LIN {X 0,Y 309.454,Z 977.493,A -85,B 0,C 180,E1 27160.011,E2 27160.011} C_VEL
LIN {X 0,Y 310.124,Z 964.953,A -85,B 0,C 180,E1 27165.897,E2 27165.897} C_VEL
LIN {X 0,Y 310.342,Z 957.233,A -85,B 0,C 180,E1 27171.598,E2 27171.598} C_VEL
LIN {X 0,Y 311.292,Z 953.109,A -85,B 0,C 180,E1 27177.214,E2 27177.214} C_VEL
LIN {X 0,Y 311.401,Z 954.291,A -85,B 0,C 180,E1 27181.386,E2 27181.386} C_VEL
LIN {X 0,Y 311.732,Z 959.799,A -85,B 0,C 180,E1 27186.955,E2 27186.955} C_VEL
LIN {X 0,Y 312.391,Z 969.833,A -85,B 0,C 180,E1 27192.716,E2 27192.716} C_VEL
LIN {X 0,Y 312.414,Z 984.77,A -85,B 0,C 180,E1 27198.53,E2 27198.53} C_VEL
LIN {X 0,Y 312.191,Z 989.255,A -85,B 0,C 180,E1 27199.981,E2 27199.981} C_VEL
LIN {X 0,Y 287.34,Z 1027.158,A -85,B 0,C 180,E1 27203.968,E2 27203.968} C_VEL
LIN {X 0,Y 260.3,Z 1061.028,A -85,B 0,C 180,E1 27209.446,E2 27209.446} C_VEL
LIN {X 0,Y 233.843,Z 1089.665,A -85,B 0,C 180,E1 27216.897,E2 27216.897} C_VEL
LIN {X 0,Y 212.045,Z 1111.278,A -85,B 0,C 180,E1 27225.984,E2 27225.984} C_VEL
LIN {X 0,Y 195.512,Z 1127.849,A -85,B 0,C 180,E1 27237.243,E2 27237.243} C_VEL
LIN {X 0,Y 185.737,Z 1139.665,A -85,B 0,C 180,E1 27251.006,E2 27251.006} C_VEL
LIN {X 0,Y 183.31,Z 1144.428,A -85,B 0,C 180,E1 27261.462,E2 27261.462} C_VEL
LIN {X 0,Y 183.515,Z 1145.902,A -85,B 0,C 180,E1 27269.997,E2 27269.997} C_VEL
LIN {X 0,Y 183.436,Z 1145.117,A -85,B 0,C 180,E1 27279.48,E2 27279.48} C_VEL
LIN {X 0,Y 186.512,Z 1140.958,A -85,B 0,C 180,E1 27290.599,E2 27290.599} C_VEL
LIN {X 0,Y 197.046,Z 1130.929,A -85,B 0,C 180,E1 27303.776,E2 27303.776} C_VEL
LIN {X 0,Y 217.166,Z 1113.725,A -85,B 0,C 180,E1 27316.111,E2 27316.111} C_VEL
LIN {X 0,Y 243.736,Z 1090.221,A -85,B 0,C 180,E1 27325.671,E2 27325.671} C_VEL
LIN {X 0,Y 272.358,Z 1061.63,A -85,B 0,C 180,E1 27332.584,E2 27332.584} C_VEL
LIN {X 0,Y 300.342,Z 1028.677,A -85,B 0,C 180,E1 27337.531,E2 27337.531} C_VEL
LIN {X 0,Y 320.87,Z 1000.29,A -85,B 0,C 180,E1 27340.365,E2 27340.365} C_VEL
LIN {X 0,Y 321.893,Z 993.539,A -85,B 0,C 180,E1 27342.656,E2 27342.656} C_VEL
LIN {X 0,Y 322.199,Z 981.849,A -85,B 0,C 180,E1 27348.504,E2 27348.504} C_VEL
LIN {X 0,Y 322.094,Z 974.677,A -85,B 0,C 180,E1 27354.621,E2 27354.621} C_VEL
LIN {X 0,Y 322.235,Z 972.945,A -85,B 0,C 180,E1 27357.317,E2 27357.317} C_VEL
LIN {X 0,Y 322.11,Z 972.654,A -85,B 0,C 180,E1 27360.004,E2 27360.004} C_VEL
LIN {X 0,Y 320.931,Z 976.591,A -85,B 0,C 180,E1 27365.407,E2 27365.407} C_VEL
LIN {X 0,Y 319.909,Z 984.239,A -85,B 0,C 180,E1 27370.893,E2 27370.893} C_VEL
LIN {X 0,Y 318.076,Z 996.337,A -85,B 0,C 180,E1 27376.563,E2 27376.563} C_VEL
LIN {X 0,Y 317.265,Z 1000.211,A -85,B 0,C 180,E1 27378.034,E2 27378.034} C_VEL
LIN {X 0,Y 295.491,Z 1029.491,A -85,B 0,C 180,E1 27381.587,E2 27381.587} C_VEL
LIN {X 0,Y 267.613,Z 1060.339,A -85,B 0,C 180,E1 27386.963,E2 27386.963} C_VEL
LIN {X 0,Y 241.205,Z 1085.273,A -85,B 0,C 180,E1 27393.896,E2 27393.896} C_VEL
LIN {X 0,Y 219.023,Z 1103.942,A -85,B 0,C 180,E1 27402.129,E2 27402.129} C_VEL
LIN {X 0,Y 199.19,Z 1119.649,A -85,B 0,C 180,E1 27413.993,E2 27413.993} C_VEL
LIN {X 0,Y 196.821,Z 1121.44,A -85,B 0,C 180,E1 27415.996,E2 27415.996} C_VEL
LIN {X 0,Y 188.409,Z 1125.457,A -85,B 0,C 180,E1 27420.414,E2 27420.414} C_VEL
LIN {X 0,Y 180.821,Z 1128.688,A -85,B 0,C 180,E1 27425.237,E2 27425.237} C_VEL
LIN {X 0,Y 176.46,Z 1132.191,A -85,B 0,C 180,E1 27435.117,E2 27435.117} C_VEL
LIN {X 0,Y 175.258,Z 1133.272,A -85,B 0,C 180,E1 27445.057,E2 27445.057} C_VEL
LIN {X 0,Y 176.038,Z 1131.933,A -85,B 0,C 180,E1 27454.927,E2 27454.927} C_VEL
LIN {X 0,Y 179.788,Z 1126.98,A -85,B 0,C 180,E1 27467.111,E2 27467.111} C_VEL
LIN {X 0,Y 191.399,Z 1115.835,A -85,B 0,C 180,E1 27480.879,E2 27480.879} C_VEL
LIN {X 0,Y 209.17,Z 1100.079,A -85,B 0,C 180,E1 27491.935,E2 27491.935} C_VEL
LIN {X 0,Y 231.682,Z 1079.475,A -85,B 0,C 180,E1 27500.765,E2 27500.765} C_VEL
LIN {X 0,Y 258.39,Z 1052.11,A -85,B 0,C 180,E1 27507.992,E2 27507.992} C_VEL
LIN {X 0,Y 285.416,Z 1019.388,A -85,B 0,C 180,E1 27513.41,E2 27513.41} C_VEL
LIN {X 0,Y 302.07,Z 995.756,A -85,B 0,C 180,E1 27516.102,E2 27516.102} C_VEL
LIN {X 0,Y 304.033,Z 986.317,A -85,B 0,C 180,E1 27519.215,E2 27519.215} C_VEL
LIN {X 0,Y 305.429,Z 973.42,A -85,B 0,C 180,E1 27524.943,E2 27524.943} C_VEL
LIN {X 0,Y 306.041,Z 964.764,A -85,B 0,C 180,E1 27530.947,E2 27530.947} C_VEL
LIN {X 0,Y 307.174,Z 959.952,A -85,B 0,C 180,E1 27537.176,E2 27537.176} C_VEL
LIN {X 0,Y 307.282,Z 961.092,A -85,B 0,C 180,E1 27541.404,E2 27541.404} C_VEL
LIN {X 0,Y 307.545,Z 967.728,A -85,B 0,C 180,E1 27547.76,E2 27547.76} C_VEL
LIN {X 0,Y 307.681,Z 978.547,A -85,B 0,C 180,E1 27553.56,E2 27553.56} C_VEL
LIN {X 0,Y 307.106,Z 992.03,A -85,B 0,C 180,E1 27558.702,E2 27558.702} C_VEL
LIN {X 0,Y 305.015,Z 996.226,A -85,B 0,C 180,E1 27559.302,E2 27559.302} C_VEL
LIN {X 0,Y 282.523,Z 1028.725,A -85,B 0,C 180,E1 27562.74,E2 27562.74} C_VEL
LIN {X 0,Y 256.385,Z 1060.564,A -85,B 0,C 180,E1 27567.857,E2 27567.857} C_VEL
LIN {X 0,Y 228.987,Z 1089.241,A -85,B 0,C 180,E1 27575.247,E2 27575.247} C_VEL
LIN {X 0,Y 206.22,Z 1110.893,A -85,B 0,C 180,E1 27584.399,E2 27584.399} C_VEL
LIN {X 0,Y 188.676,Z 1127.497,A -85,B 0,C 180,E1 27595.897,E2 27595.897} C_VEL
LIN {X 0,Y 178.135,Z 1139.34,A -85,B 0,C 180,E1 27610.162,E2 27610.162} C_VEL
LIN {X 0,Y 175.558,Z 1143.769,A -85,B 0,C 180,E1 27620.084,E2 27620.084} C_VEL
LIN {X 0,Y 175.605,Z 1145.616,A -85,B 0,C 180,E1 27629.997,E2 27629.997} C_VEL
LIN {X 0,Y 175.561,Z 1144.846,A -85,B 0,C 180,E1 27639.91,E2 27639.91} C_VEL
LIN {X 0,Y 179.205,Z 1140.454,A -85,B 0,C 180,E1 27651.988,E2 27651.988} C_VEL
LIN {X 0,Y 190.306,Z 1130.7,A -85,B 0,C 180,E1 27665.144,E2 27665.144} C_VEL
LIN {X 0,Y 210.651,Z 1114.288,A -85,B 0,C 180,E1 27677.288,E2 27677.288} C_VEL
LIN {X 0,Y 237.393,Z 1091.652,A -85,B 0,C 180,E1 27686.769,E2 27686.769} C_VEL
LIN {X 0,Y 265.849,Z 1064.402,A -85,B 0,C 180,E1 27693.552,E2 27693.552} C_VEL
LIN {X 0,Y 292.81,Z 1034.247,A -85,B 0,C 180,E1 27698.264,E2 27698.264} C_VEL
LIN {X 0,Y 316.359,Z 1002.822,A -85,B 0,C 180,E1 27701.561,E2 27701.561} C_VEL
LIN {X 0,Y 317.281,Z 991.089,A -85,B 0,C 180,E1 27706.932,E2 27706.932} C_VEL
LIN {X 0,Y 317.494,Z 984.09,A -85,B 0,C 180,E1 27711.797,E2 27711.797} C_VEL
LIN {X 0,Y 317.754,Z 979.539,A -85,B 0,C 180,E1 27717.279,E2 27717.279} C_VEL
LIN {X 0,Y 317.364,Z 979.71,A -85,B 0,C 180,E1 27720.922,E2 27720.922} C_VEL
LIN {X 0,Y 315.966,Z 984.954,A -85,B 0,C 180,E1 27727.008,E2 27727.008} C_VEL
LIN {X 0,Y 314.446,Z 993.783,A -85,B 0,C 180,E1 27732.491,E2 27732.491} C_VEL
LIN {X 0,Y 312.348,Z 1003.618,A -85,B 0,C 180,E1 27736.876,E2 27736.876} C_VEL
LIN {X 0,Y 310.356,Z 1006.988,A -85,B 0,C 180,E1 27737.456,E2 27737.456} C_VEL
LIN {X 0,Y 281.848,Z 1041.952,A -85,B 0,C 180,E1 27741.953,E2 27741.953} C_VEL
LIN {X 0,Y 251.952,Z 1072.057,A -85,B 0,C 180,E1 27748.147,E2 27748.147} C_VEL
LIN {X 0,Y 224.69,Z 1095.458,A -85,B 0,C 180,E1 27756.196,E2 27756.196} C_VEL
LIN {X 0,Y 201.8,Z 1112.987,A -85,B 0,C 180,E1 27766.417,E2 27766.417} C_VEL
LIN {X 0,Y 186.729,Z 1124.294,A -85,B 0,C 180,E1 27777.828,E2 27777.828} C_VEL
LIN {X 0,Y 180.821,Z 1128.688,A -85,B 0,C 180,E1 27785.237,E2 27785.237} C_VEL
LIN {X 0,Y 176.154,Z 1130.599,A -85,B 0,C 180,E1 27789.115,E2 27789.115} C_VEL
LIN {X 0,Y 168.559,Z 1132.598,A -85,B 0,C 180,E1 27795.169,E2 27795.169} C_VEL
LIN {X 0,Y 168.269,Z 1132.704,A -85,B 0,C 180,E1 27795.909,E2 27795.909} C_VEL
LIN {X 0,Y 167.345,Z 1133.56,A -85,B 0,C 180,E1 27804.822,E2 27804.822} C_VEL
LIN {X 0,Y 168.161,Z 1132.229,A -85,B 0,C 180,E1 27815.159,E2 27815.159} C_VEL
LIN {X 0,Y 172.214,Z 1127.308,A -85,B 0,C 180,E1 27827.888,E2 27827.888} C_VEL
LIN {X 0,Y 184.575,Z 1116.187,A -85,B 0,C 180,E1 27842.154,E2 27842.154} C_VEL
LIN {X 0,Y 203.287,Z 1100.465,A -85,B 0,C 180,E1 27853.443,E2 27853.443} C_VEL
LIN {X 0,Y 226.708,Z 1079.898,A -85,B 0,C 180,E1 27862.331,E2 27862.331} C_VEL
LIN {X 0,Y 253.939,Z 1052.898,A -85,B 0,C 180,E1 27869.445,E2 27869.445} C_VEL
LIN {X 0,Y 281.772,Z 1020.113,A -85,B 0,C 180,E1 27874.823,E2 27874.823} C_VEL
LIN {X 0,Y 297.696,Z 997.877,A -85,B 0,C 180,E1 27877.424,E2 27877.424} C_VEL
LIN {X 0,Y 300.165,Z 983.944,A -85,B 0,C 180,E1 27883.045,E2 27883.045} C_VEL
LIN {X 0,Y 301.3,Z 974.505,A -85,B 0,C 180,E1 27888.425,E2 27888.425} C_VEL
LIN {X 0,Y 302.298,Z 968.507,A -85,B 0,C 180,E1 27894.259,E2 27894.259} C_VEL
LIN {X 0,Y 302.991,Z 966.741,A -85,B 0,C 180,E1 27897.137,E2 27897.137} C_VEL
LIN {X 0,Y 303.1,Z 967.874,A -85,B 0,C 180,E1 27901.424,E2 27901.424} C_VEL
LIN {X 0,Y 303.108,Z 974.62,A -85,B 0,C 180,E1 27907.874,E2 27907.874} C_VEL
LIN {X 0,Y 302.846,Z 985.681,A -85,B 0,C 180,E1 27913.703,E2 27913.703} C_VEL
LIN {X 0,Y 301.796,Z 996.683,A -85,B 0,C 180,E1 27917.943,E2 27917.943} C_VEL
LIN {X 0,Y 277.843,Z 1030.29,A -85,B 0,C 180,E1 27921.47,E2 27921.47} C_VEL
LIN {X 0,Y 250.98,Z 1061.929,A -85,B 0,C 180,E1 27926.585,E2 27926.585} C_VEL
LIN {X 0,Y 223.105,Z 1090.047,A -85,B 0,C 180,E1 27933.928,E2 27933.928} C_VEL
LIN {X 0,Y 197.761,Z 1113.049,A -85,B 0,C 180,E1 27944.125,E2 27944.125} C_VEL
LIN {X 0,Y 179.941,Z 1129.015,A -85,B 0,C 180,E1 27956.302,E2 27956.302} C_VEL
LIN {X 0,Y 170.58,Z 1139.013,A -85,B 0,C 180,E1 27969.244,E2 27969.244} C_VEL
LIN {X 0,Y 167.367,Z 1144.369,A -85,B 0,C 180,E1 27983.143,E2 27983.143} C_VEL
LIN {X 0,Y 167.695,Z 1145.33,A -85,B 0,C 180,E1 27989.997,E2 27989.997} C_VEL
LIN {X 0,Y 167.704,Z 1144.576,A -85,B 0,C 180,E1 28000.379,E2 28000.379} C_VEL
LIN {X 0,Y 173.437,Z 1138.737,A -85,B 0,C 180,E1 28015.823,E2 28015.823} C_VEL
LIN {X 0,Y 188.304,Z 1126.942,A -85,B 0,C 180,E1 28029.936,E2 28029.936} C_VEL
LIN {X 0,Y 209.62,Z 1110.564,A -85,B 0,C 180,E1 28040.796,E2 28040.796} C_VEL
LIN {X 0,Y 236.369,Z 1088.569,A -85,B 0,C 180,E1 28049.353,E2 28049.353} C_VEL
LIN {X 0,Y 266.452,Z 1060.199,A -85,B 0,C 180,E1 28055.909,E2 28055.909} C_VEL
LIN {X 0,Y 296.399,Z 1026.341,A -85,B 0,C 180,E1 28060.667,E2 28060.667} C_VEL
LIN {X 0,Y 311.26,Z 1006.345,A -85,B 0,C 180,E1 28062.709,E2 28062.709} C_VEL
LIN {X 0,Y 312.419,Z 995.821,A -85,B 0,C 180,E1 28067.932,E2 28067.932} C_VEL
LIN {X 0,Y 312.75,Z 989.184,A -85,B 0,C 180,E1 28073.068,E2 28073.068} C_VEL
LIN {X 0,Y 313.176,Z 986.028,A -85,B 0,C 180,E1 28077.239,E2 28077.239} C_VEL
LIN {X 0,Y 313.053,Z 985.699,A -85,B 0,C 180,E1 28080.004,E2 28080.004} C_VEL
LIN {X 0,Y 311.462,Z 989.786,A -85,B 0,C 180,E1 28085.572,E2 28085.572} C_VEL
LIN {X 0,Y 309.922,Z 996.772,A -85,B 0,C 180,E1 28090.639,E2 28090.639} C_VEL
LIN {X 0,Y 307.308,Z 1007.696,A -85,B 0,C 180,E1 28095.956,E2 28095.956} C_VEL
LIN {X 0,Y 279.608,Z 1041.247,A -85,B 0,C 180,E1 28100.273,E2 28100.273} C_VEL
LIN {X 0,Y 249.573,Z 1070.924,A -85,B 0,C 180,E1 28106.175,E2 28106.175} C_VEL
LIN {X 0,Y 221.618,Z 1094.277,A -85,B 0,C 180,E1 28113.878,E2 28113.878} C_VEL
LIN {X 0,Y 199.18,Z 1110.983,A -85,B 0,C 180,E1 28123.062,E2 28123.062} C_VEL
LIN {X 0,Y 179.996,Z 1124.437,A -85,B 0,C 180,E1 28136.312,E2 28136.312} C_VEL
LIN {X 0,Y 170.661,Z 1131.02,A -85,B 0,C 180,E1 28149.26,E2 28149.26} C_VEL
LIN {X 0,Y 168.269,Z 1132.704,A -85,B 0,C 180,E1 28155.909,E2 28155.909} C_VEL
LIN {X 0,Y 164.949,Z 1133.468,A -85,B 0,C 180,E1 28160.259,E2 28160.259} C_VEL
LIN {X 0,Y 159.505,Z 1133.688,A -85,B 0,C 180,E1 28167.01,E2 28167.01} C_VEL
LIN {X 0,Y 159.476,Z 1133.631,A -85,B 0,C 180,E1 28167.801,E2 28167.801} C_VEL
LIN {X 0,Y 160.307,Z 1132.525,A -85,B 0,C 180,E1 28175.412,E2 28175.412} C_VEL
LIN {X 0,Y 164.681,Z 1127.635,A -85,B 0,C 180,E1 28188.736,E2 28188.736} C_VEL
LIN {X 0,Y 177.847,Z 1116.538,A -85,B 0,C 180,E1 28203.527,E2 28203.527} C_VEL
LIN {X 0,Y 197.547,Z 1100.85,A -85,B 0,C 180,E1 28215.041,E2 28215.041} C_VEL
LIN {X 0,Y 223.181,Z 1079.148,A -85,B 0,C 180,E1 28224.344,E2 28224.344} C_VEL
LIN {X 0,Y 251.638,Z 1051.584,A -85,B 0,C 180,E1 28231.376,E2 28231.376} C_VEL
LIN {X 0,Y 280.049,Z 1018.714,A -85,B 0,C 180,E1 28236.538,E2 28236.538} C_VEL
LIN {X 0,Y 292.521,Z 1001.831,A -85,B 0,C 180,E1 28238.415,E2 28238.415} C_VEL
LIN {X 0,Y 295.236,Z 989.526,A -85,B 0,C 180,E1 28243.545,E2 28243.545} C_VEL
LIN {X 0,Y 296.655,Z 981.453,A -85,B 0,C 180,E1 28248.241,E2 28248.241} C_VEL
LIN {X 0,Y 297.788,Z 975.178,A -85,B 0,C 180,E1 28254.172,E2 28254.172} C_VEL
LIN {X 0,Y 298.613,Z 973.397,A -85,B 0,C 180,E1 28257.095,E2 28257.095} C_VEL
LIN {X 0,Y 298.705,Z 974.518,A -85,B 0,C 180,E1 28261.445,E2 28261.445} C_VEL
LIN {X 0,Y 298.49,Z 981.466,A -85,B 0,C 180,E1 28267.997,E2 28267.997} C_VEL
LIN {X 0,Y 297.701,Z 992.509,A -85,B 0,C 180,E1 28273.806,E2 28273.806} C_VEL
LIN {X 0,Y 296.878,Z 999.978,A -85,B 0,C 180,E1 28276.765,E2 28276.765} C_VEL
LIN {X 0,Y 268.977,Z 1037.272,A -85,B 0,C 180,E1 28280.878,E2 28280.878} C_VEL
LIN {X 0,Y 240.531,Z 1068.562,A -85,B 0,C 180,E1 28286.402,E2 28286.402} C_VEL
LIN {X 0,Y 214.164,Z 1093.626,A -85,B 0,C 180,E1 28293.59,E2 28293.59} C_VEL
LIN {X 0,Y 190.431,Z 1114.141,A -85,B 0,C 180,E1 28303.245,E2 28303.245} C_VEL
LIN {X 0,Y 171.503,Z 1130.225,A -85,B 0,C 180,E1 28316.419,E2 28316.419} C_VEL
LIN {X 0,Y 161.893,Z 1139.987,A -85,B 0,C 180,E1 28330.929,E2 28330.929} C_VEL
LIN {X 0,Y 159.495,Z 1144.421,A -85,B 0,C 180,E1 28344.56,E2 28344.56} C_VEL
LIN {X 0,Y 159.797,Z 1145.045,A -85,B 0,C 180,E1 28349.997,E2 28349.997} C_VEL
LIN {X 0,Y 159.842,Z 1144.304,A -85,B 0,C 180,E1 28360.896,E2 28360.896} C_VEL
LIN {X 0,Y 166.167,Z 1138.49,A -85,B 0,C 180,E1 28377.042,E2 28377.042} C_VEL
LIN {X 0,Y 183.695,Z 1125.645,A -85,B 0,C 180,E1 28392.573,E2 28392.573} C_VEL
LIN {X 0,Y 209.582,Z 1106.659,A -85,B 0,C 180,E1 28404.386,E2 28404.386} C_VEL
LIN {X 0,Y 239.72,Z 1082.029,A -85,B 0,C 180,E1 28412.847,E2 28412.847} C_VEL
LIN {X 0,Y 269.467,Z 1053.611,A -85,B 0,C 180,E1 28418.583,E2 28418.583} C_VEL
LIN {X 0,Y 296.724,Z 1022.644,A -85,B 0,C 180,E1 28422.514,E2 28422.514} C_VEL
LIN {X 0,Y 306.171,Z 1010.273,A -85,B 0,C 180,E1 28423.751,E2 28423.751} C_VEL
LIN {X 0,Y 307.598,Z 1000.079,A -85,B 0,C 180,E1 28429.262,E2 28429.262} C_VEL
LIN {X 0,Y 308.074,Z 994.353,A -85,B 0,C 180,E1 28434.376,E2 28434.376} C_VEL
LIN {X 0,Y 308.402,Z 992.413,A -85,B 0,C 180,E1 28437.196,E2 28437.196} C_VEL
LIN {X 0,Y 308.295,Z 992.056,A -85,B 0,C 180,E1 28440.004,E2 28440.004} C_VEL
LIN {X 0,Y 306.568,Z 996.274,A -85,B 0,C 180,E1 28445.661,E2 28445.661} C_VEL
LIN {X 0,Y 304.544,Z 1003.435,A -85,B 0,C 180,E1 28450.829,E2 28450.829} C_VEL
LIN {X 0,Y 302.291,Z 1011.366,A -85,B 0,C 180,E1 28454.846,E2 28454.846} C_VEL
LIN {X 0,Y 275.542,Z 1042.801,A -85,B 0,C 180,E1 28458.919,E2 28458.919} C_VEL
LIN {X 0,Y 244.948,Z 1072.087,A -85,B 0,C 180,E1 28464.72,E2 28464.72} C_VEL
LIN {X 0,Y 215.386,Z 1095.811,A -85,B 0,C 180,E1 28472.663,E2 28472.663} C_VEL
LIN {X 0,Y 191.129,Z 1112.845,A -85,B 0,C 180,E1 28482.57,E2 28482.57} C_VEL
LIN {X 0,Y 171.669,Z 1125.654,A -85,B 0,C 180,E1 28496.367,E2 28496.367} C_VEL
LIN {X 0,Y 163.133,Z 1131.282,A -85,B 0,C 180,E1 28508.256,E2 28508.256} C_VEL
LIN {X 0,Y 159.816,Z 1133.583,A -85,B 0,C 180,E1 28519.103,E2 28519.103} C_VEL
LIN {X 0,Y 159.476,Z 1133.631,A -85,B 0,C 180,E1 28527.801,E2 28527.801} C_VEL
LIN {X 0,Y 157.366,Z 1133.201,A -85,B 0,C 180,E1 28532.48,E2 28532.48} C_VEL
LIN {X 0,Y 153.389,Z 1131.539,A -85,B 0,C 180,E1 28540.523,E2 28540.523} C_VEL
LIN {X 0,Y 160.85,Z 1124.949,A -85,B 0,C 180,E1 28555.012,E2 28555.012} C_VEL
LIN {X 0,Y 179.309,Z 1110.927,A -85,B 0,C 180,E1 28570.312,E2 28570.312} C_VEL
LIN {X 0,Y 204.992,Z 1091.025,A -85,B 0,C 180,E1 28581.773,E2 28581.773} C_VEL
LIN {X 0,Y 233.615,Z 1066.025,A -85,B 0,C 180,E1 28589.903,E2 28589.903} C_VEL
LIN {X 0,Y 261.479,Z 1037.424,A -85,B 0,C 180,E1 28595.538,E2 28595.538} C_VEL
LIN {X 0,Y 287.755,Z 1004.894,A -85,B 0,C 180,E1 28599.73,E2 28599.73} C_VEL
LIN {X 0,Y 290.688,Z 993.375,A -85,B 0,C 180,E1 28604.933,E2 28604.933} C_VEL
LIN {X 0,Y 292.054,Z 986.379,A -85,B 0,C 180,E1 28609.452,E2 28609.452} C_VEL
LIN {X 0,Y 293.263,Z 981.857,A -85,B 0,C 180,E1 28614.081,E2 28614.081} C_VEL
LIN {X 0,Y 294.123,Z 979.999,A -85,B 0,C 180,E1 28617.051,E2 28617.051} C_VEL
LIN {X 0,Y 294.203,Z 981.13,A -85,B 0,C 180,E1 28621.467,E2 28621.467} C_VEL
LIN {X 0,Y 293.788,Z 987.176,A -85,B 0,C 180,E1 28627.382,E2 28627.382} C_VEL
LIN {X 0,Y 292.679,Z 997.658,A -85,B 0,C 180,E1 28633.146,E2 28633.146} C_VEL
LIN {X 0,Y 291.155,Z 1004.413,A -85,B 0,C 180,E1 28635.725,E2 28635.725} C_VEL
LIN {X 0,Y 264.513,Z 1038.724,A -85,B 0,C 180,E1 28639.505,E2 28639.505} C_VEL
LIN {X 0,Y 234.012,Z 1071.132,A -85,B 0,C 180,E1 28645.301,E2 28645.301} C_VEL
LIN {X 0,Y 204.459,Z 1097.801,A -85,B 0,C 180,E1 28653.445,E2 28653.445} C_VEL
LIN {X 0,Y 179.421,Z 1118.05,A -85,B 0,C 180,E1 28664.281,E2 28664.281} C_VEL
LIN {X 0,Y 163.219,Z 1131.213,A -85,B 0,C 180,E1 28676.403,E2 28676.403} C_VEL
LIN {X 0,Y 153.311,Z 1140.929,A -85,B 0,C 180,E1 28692.797,E2 28692.797} C_VEL
LIN {X 0,Y 151.573,Z 1144.313,A -85,B 0,C 180,E1 28705.293,E2 28705.293} C_VEL
LIN {X 0,Y 151.885,Z 1144.758,A -85,B 0,C 180,E1 28709.997,E2 28709.997} C_VEL
LIN {X 0,Y 151.992,Z 1144.033,A -85,B 0,C 180,E1 28721.466,E2 28721.466} C_VEL
LIN {X 0,Y 158.972,Z 1138.242,A -85,B 0,C 180,E1 28738.374,E2 28738.374} C_VEL
LIN {X 0,Y 177.932,Z 1125.291,A -85,B 0,C 180,E1 28754.474,E2 28754.474} C_VEL
LIN {X 0,Y 204.928,Z 1106.462,A -85,B 0,C 180,E1 28766.245,E2 28766.245} C_VEL
LIN {X 0,Y 235.976,Z 1081.975,A -85,B 0,C 180,E1 28774.584,E2 28774.584} C_VEL
LIN {X 0,Y 266.743,Z 1053.386,A -85,B 0,C 180,E1 28780.211,E2 28780.211} C_VEL
LIN {X 0,Y 294.9,Z 1021.977,A -85,B 0,C 180,E1 28784.059,E2 28784.059} C_VEL
LIN {X 0,Y 300.558,Z 1014.903,A -85,B 0,C 180,E1 28784.709,E2 28784.709} C_VEL
LIN {X 0,Y 302.199,Z 1007.532,A -85,B 0,C 180,E1 28788.469,E2 28788.469} C_VEL
LIN {X 0,Y 303.117,Z 1000.705,A -85,B 0,C 180,E1 28794.283,E2 28794.283} C_VEL
LIN {X 0,Y 303.553,Z 998.736,A -85,B 0,C 180,E1 28797.151,E2 28797.151} C_VEL
LIN {X 0,Y 303.444,Z 998.357,A -85,B 0,C 180,E1 28800.004,E2 28800.004} C_VEL
LIN {X 0,Y 301.4,Z 1002.596,A -85,B 0,C 180,E1 28805.758,E2 28805.758} C_VEL
LIN {X 0,Y 299.096,Z 1009.843,A -85,B 0,C 180,E1 28810.924,E2 28810.924} C_VEL
LIN {X 0,Y 296.838,Z 1015.991,A -85,B 0,C 180,E1 28813.963,E2 28813.963} C_VEL
LIN {X 0,Y 268.444,Z 1047.426,A -85,B 0,C 180,E1 28818.012,E2 28818.012} C_VEL
LIN {X 0,Y 238.959,Z 1074.455,A -85,B 0,C 180,E1 28823.523,E2 28823.523} C_VEL
LIN {X 0,Y 208.498,Z 1097.898,A -85,B 0,C 180,E1 28831.62,E2 28831.62} C_VEL
LIN {X 0,Y 181.1,Z 1116.016,A -85,B 0,C 180,E1 28843.109,E2 28843.109} C_VEL
LIN {X 0,Y 163.446,Z 1126.781,A -85,B 0,C 180,E1 28856.312,E2 28856.312} C_VEL
LIN {X 0,Y 155.668,Z 1131.544,A -85,B 0,C 180,E1 28867.155,E2 28867.155} C_VEL
LIN {X 0,Y 151.976,Z 1133.863,A -85,B 0,C 180,E1 28878.533,E2 28878.533} C_VEL
LIN {X 0,Y 151.876,Z 1133.769,A -85,B 0,C 180,E1 28890.003,E2 28890.003} C_VEL
LIN {X 0,Y 153.389,Z 1131.539,A -85,B 0,C 180,E1 28900.523,E2 28900.523} C_VEL
LIN {X 0,Y 152.567,Z 1130.067,A -85,B 0,C 180,E1 28905.395,E2 28905.395} C_VEL
LIN {X 0,Y 151.111,Z 1127.164,A -85,B 0,C 180,E1 28912.806,E2 28912.806} C_VEL
LIN {X 0,Y 151.569,Z 1126.738,A -85,B 0,C 180,E1 28913.607,E2 28913.607} C_VEL
LIN {X 0,Y 166.471,Z 1116.088,A -85,B 0,C 180,E1 28927.79,E2 28927.79} C_VEL
LIN {X 0,Y 191.243,Z 1098.244,A -85,B 0,C 180,E1 28940.393,E2 28940.393} C_VEL
LIN {X 0,Y 219.933,Z 1075.178,A -85,B 0,C 180,E1 28949.287,E2 28949.287} C_VEL
LIN {X 0,Y 249.039,Z 1047.712,A -85,B 0,C 180,E1 28955.532,E2 28955.532} C_VEL
LIN {X 0,Y 276.837,Z 1016.283,A -85,B 0,C 180,E1 28959.966,E2 28959.966} C_VEL
LIN {X 0,Y 282.705,Z 1008.809,A -85,B 0,C 180,E1 28960.767,E2 28960.767} C_VEL
LIN {X 0,Y 285.99,Z 997.519,A -85,B 0,C 180,E1 28966.243,E2 28966.243} C_VEL
LIN {X 0,Y 287.558,Z 991.171,A -85,B 0,C 180,E1 28970.926,E2 28970.926} C_VEL
LIN {X 0,Y 289.464,Z 986.5,A -85,B 0,C 180,E1 28977.004,E2 28977.004} C_VEL
LIN {X 0,Y 289.808,Z 986.58,A -85,B 0,C 180,E1 28979.995,E2 28979.995} C_VEL
LIN {X 0,Y 288.97,Z 992.469,A -85,B 0,C 180,E1 28986.489,E2 28986.489} C_VEL
LIN {X 0,Y 287.693,Z 1001.94,A -85,B 0,C 180,E1 28992.121,E2 28992.121} C_VEL
LIN {X 0,Y 286.123,Z 1007.881,A -85,B 0,C 180,E1 28994.501,E2 28994.501} C_VEL
LIN {X 0,Y 260.298,Z 1040.017,A -85,B 0,C 180,E1 28998.076,E2 28998.076} C_VEL
LIN {X 0,Y 230.622,Z 1070.691,A -85,B 0,C 180,E1 29003.457,E2 29003.457} C_VEL
LIN {X 0,Y 199.629,Z 1097.744,A -85,B 0,C 180,E1 29011.616,E2 29011.616} C_VEL
LIN {X 0,Y 171.756,Z 1119.251,A -85,B 0,C 180,E1 29023.458,E2 29023.458} C_VEL
LIN {X 0,Y 153.785,Z 1132.963,A -85,B 0,C 180,E1 29037.599,E2 29037.599} C_VEL
LIN {X 0,Y 145.634,Z 1140.611,A -85,B 0,C 180,E1 29051.86,E2 29051.86} C_VEL
LIN {X 0,Y 143.683,Z 1143.828,A -85,B 0,C 180,E1 29063.96,E2 29063.96} C_VEL
LIN {X 0,Y 143.99,Z 1144.473,A -85,B 0,C 180,E1 29069.997,E2 29069.997} C_VEL
LIN {X 0,Y 144.154,Z 1143.762,A -85,B 0,C 180,E1 29082.098,E2 29082.098} C_VEL
LIN {X 0,Y 149.855,Z 1139.278,A -85,B 0,C 180,E1 29096.982,E2 29096.982} C_VEL
LIN {X 0,Y 165.641,Z 1129.157,A -85,B 0,C 180,E1 29112.339,E2 29112.339} C_VEL
LIN {X 0,Y 190.049,Z 1113.415,A -85,B 0,C 180,E1 29124.582,E2 29124.582} C_VEL
LIN {X 0,Y 220.849,Z 1091.221,A -85,B 0,C 180,E1 29133.781,E2 29133.781} C_VEL
LIN {X 0,Y 251.441,Z 1065.375,A -85,B 0,C 180,E1 29139.883,E2 29139.883} C_VEL
LIN {X 0,Y 280.77,Z 1035.852,A -85,B 0,C 180,E1 29144.154,E2 29144.154} C_VEL
LIN {X 0,Y 295.912,Z 1017.976,A -85,B 0,C 180,E1 29145.983,E2 29145.983} C_VEL
LIN {X 0,Y 297.562,Z 1009.915,A -85,B 0,C 180,E1 29151.243,E2 29151.243} C_VEL
LIN {X 0,Y 298.495,Z 1004.901,A -85,B 0,C 180,E1 29157.103,E2 29157.103} C_VEL
LIN {X 0,Y 298.388,Z 1004.512,A -85,B 0,C 180,E1 29160.004,E2 29160.004} C_VEL
LIN {X 0,Y 296.22,Z 1008.895,A -85,B 0,C 180,E1 29165.859,E2 29165.859} C_VEL
LIN {X 0,Y 293.539,Z 1015.851,A -85,B 0,C 180,E1 29170.867,E2 29170.867} C_VEL
LIN {X 0,Y 292.528,Z 1018.645,A -85,B 0,C 180,E1 29172.383,E2 29172.383} C_VEL
LIN {X 0,Y 289.598,Z 1022.431,A -85,B 0,C 180,E1 29173.091,E2 29173.091} C_VEL
LIN {X 0,Y 259.377,Z 1054.051,A -85,B 0,C 180,E1 29177.401,E2 29177.401} C_VEL
LIN {X 0,Y 227.416,Z 1081.247,A -85,B 0,C 180,E1 29183.498,E2 29183.498} C_VEL
LIN {X 0,Y 196.472,Z 1103.223,A -85,B 0,C 180,E1 29192.222,E2 29192.222} C_VEL
LIN {X 0,Y 171.543,Z 1118.53,A -85,B 0,C 180,E1 29203.391,E2 29203.391} C_VEL
LIN {X 0,Y 154.01,Z 1128.642,A -85,B 0,C 180,E1 29217.59,E2 29217.59} C_VEL
LIN {X 0,Y 145.64,Z 1133.274,A -85,B 0,C 180,E1 29231.868,E2 29231.868} C_VEL
LIN {X 0,Y 143.623,Z 1134.421,A -85,B 0,C 180,E1 29243.964,E2 29243.964} C_VEL
LIN {X 0,Y 144.57,Z 1133.117,A -85,B 0,C 180,E1 29256.003,E2 29256.003} C_VEL
LIN {X 0,Y 149.7,Z 1128.292,A -85,B 0,C 180,E1 29270.693,E2 29270.693} C_VEL
LIN {X 0,Y 151.569,Z 1126.738,A -85,B 0,C 180,E1 29273.607,E2 29273.607} C_VEL
LIN {X 0,Y 152.888,Z 1123.407,A -85,B 0,C 180,E1 29280.066,E2 29280.066} C_VEL
LIN {X 0,Y 155.714,Z 1119.342,A -85,B 0,C 180,E1 29286.334,E2 29286.334} C_VEL
LIN {X 0,Y 179.01,Z 1103.694,A -85,B 0,C 180,E1 29299.445,E2 29299.445} C_VEL
LIN {X 0,Y 208.711,Z 1081.588,A -85,B 0,C 180,E1 29309.296,E2 29309.296} C_VEL
LIN {X 0,Y 240.432,Z 1053.651,A -85,B 0,C 180,E1 29316.241,E2 29316.241} C_VEL
LIN {X 0,Y 271.466,Z 1020.221,A -85,B 0,C 180,E1 29321.143,E2 29321.143} C_VEL
LIN {X 0,Y 278.037,Z 1011.698,A -85,B 0,C 180,E1 29322.261,E2 29322.261} C_VEL
LIN {X 0,Y 281.332,Z 1001.712,A -85,B 0,C 180,E1 29327.591,E2 29327.591} C_VEL
LIN {X 0,Y 283.629,Z 994.843,A -85,B 0,C 180,E1 29333.88,E2 29333.88} C_VEL
LIN {X 0,Y 284.658,Z 992.922,A -85,B 0,C 180,E1 29336.953,E2 29336.953} C_VEL
LIN {X 0,Y 285.025,Z 992.963,A -85,B 0,C 180,E1 29339.995,E2 29339.995} C_VEL
LIN {X 0,Y 284.021,Z 999.036,A -85,B 0,C 180,E1 29346.602,E2 29346.602} C_VEL
LIN {X 0,Y 282.151,Z 1008.834,A -85,B 0,C 180,E1 29352.363,E2 29352.363} C_VEL
LIN {X 0,Y 281.384,Z 1011.19,A -85,B 0,C 180,E1 29353.249,E2 29353.249} C_VEL
LIN {X 0,Y 252.961,Z 1044.88,A -85,B 0,C 180,E1 29357.095,E2 29357.095} C_VEL
LIN {X 0,Y 224.418,Z 1072.963,A -85,B 0,C 180,E1 29362.197,E2 29362.197} C_VEL
LIN {X 0,Y 194.097,Z 1098.374,A -85,B 0,C 180,E1 29369.985,E2 29369.985} C_VEL
LIN {X 0,Y 166.233,Z 1118.877,A -85,B 0,C 180,E1 29381.41,E2 29381.41} C_VEL
LIN {X 0,Y 146.376,Z 1133.094,A -85,B 0,C 180,E1 29396.58,E2 29396.58} C_VEL
LIN {X 0,Y 138.023,Z 1140.293,A -85,B 0,C 180,E1 29410.822,E2 29410.822} C_VEL
LIN {X 0,Y 135.797,Z 1143.532,A -85,B 0,C 180,E1 29423.607,E2 29423.607} C_VEL
LIN {X 0,Y 135.963,Z 1144.22,A -85,B 0,C 180,E1 29430.711,E2 29430.711} C_VEL
LIN {X 0,Y 136.34,Z 1143.49,A -85,B 0,C 180,E1 29442.803,E2 29442.803} C_VEL
LIN {X 0,Y 144.873,Z 1137.742,A -85,B 0,C 180,E1 29461.431,E2 29461.431} C_VEL
LIN {X 0,Y 166.662,Z 1124.844,A -85,B 0,C 180,E1 29478.414,E2 29478.414} C_VEL
LIN {X 0,Y 196.282,Z 1106.101,A -85,B 0,C 180,E1 29490.195,E2 29490.195} C_VEL
LIN {X 0,Y 228.148,Z 1082.679,A -85,B 0,C 180,E1 29498.007,E2 29498.007} C_VEL
LIN {X 0,Y 258.857,Z 1055.925,A -85,B 0,C 180,E1 29503.145,E2 29503.145} C_VEL
LIN {X 0,Y 289.546,Z 1023.51,A -85,B 0,C 180,E1 29506.958,E2 29506.958} C_VEL
LIN {X 0,Y 290.96,Z 1021.261,A -85,B 0,C 180,E1 29507.52,E2 29507.52} C_VEL
LIN {X 0,Y 292.455,Z 1014.515,A -85,B 0,C 180,E1 29512.581,E2 29512.581} C_VEL
LIN {X 0,Y 293.399,Z 1011.025,A -85,B 0,C 180,E1 29517.053,E2 29517.053} C_VEL
LIN {X 0,Y 293.289,Z 1010.619,A -85,B 0,C 180,E1 29520.005,E2 29520.005} C_VEL
LIN {X 0,Y 290.755,Z 1014.999,A -85,B 0,C 180,E1 29525.97,E2 29525.97} C_VEL
LIN {X 0,Y 287.473,Z 1022.695,A -85,B 0,C 180,E1 29531.314,E2 29531.314} C_VEL
LIN {X 0,Y 283.735,Z 1027.099,A -85,B 0,C 180,E1 29532.011,E2 29532.011} C_VEL
LIN {X 0,Y 254.263,Z 1056.637,A -85,B 0,C 180,E1 29536.099,E2 29536.099} C_VEL
LIN {X 0,Y 223.256,Z 1082.204,A -85,B 0,C 180,E1 29541.808,E2 29541.808} C_VEL
LIN {X 0,Y 192.223,Z 1103.413,A -85,B 0,C 180,E1 29550.153,E2 29550.153} C_VEL
LIN {X 0,Y 166.035,Z 1118.754,A -85,B 0,C 180,E1 29561.341,E2 29561.341} C_VEL
LIN {X 0,Y 148.472,Z 1128.16,A -85,B 0,C 180,E1 29574.512,E2 29574.512} C_VEL
LIN {X 0,Y 138.047,Z 1133.545,A -85,B 0,C 180,E1 29590.833,E2 29590.833} C_VEL
LIN {X 0,Y 135.716,Z 1134.705,A -85,B 0,C 180,E1 29603.611,E2 29603.611} C_VEL
LIN {X 0,Y 136.713,Z 1133.413,A -85,B 0,C 180,E1 29616.35,E2 29616.35} C_VEL
LIN {X 0,Y 142.29,Z 1128.62,A -85,B 0,C 180,E1 29631.824,E2 29631.824} C_VEL
LIN {X 0,Y 155.714,Z 1119.342,A -85,B 0,C 180,E1 29646.334,E2 29646.334} C_VEL
LIN {X 0,Y 160.065,Z 1114.74,A -85,B 0,C 180,E1 29652.272,E2 29652.272} C_VEL
LIN {X 0,Y 165.698,Z 1109.423,A -85,B 0,C 180,E1 29657.821,E2 29657.821} C_VEL
LIN {X 0,Y 194.827,Z 1089.47,A -85,B 0,C 180,E1 29668.563,E2 29668.563} C_VEL
LIN {X 0,Y 227.192,Z 1063.378,A -85,B 0,C 180,E1 29676.146,E2 29676.146} C_VEL
LIN {X 0,Y 259.41,Z 1031.625,A -85,B 0,C 180,E1 29681.465,E2 29681.465} C_VEL
LIN {X 0,Y 271.939,Z 1017.172,A -85,B 0,C 180,E1 29683.121,E2 29683.121} C_VEL
LIN {X 0,Y 273.569,Z 1014.397,A -85,B 0,C 180,E1 29683.965,E2 29683.965} C_VEL
LIN {X 0,Y 276.819,Z 1005.673,A -85,B 0,C 180,E1 29689.301,E2 29689.301} C_VEL
LIN {X 0,Y 278.526,Z 1001.185,A -85,B 0,C 180,E1 29693.767,E2 29693.767} C_VEL
LIN {X 0,Y 279.715,Z 999.261,A -85,B 0,C 180,E1 29696.899,E2 29696.899} C_VEL
LIN {X 0,Y 280.139,Z 999.268,A -85,B 0,C 180,E1 29699.995,E2 29699.995} C_VEL
LIN {X 0,Y 278.758,Z 1005.759,A -85,B 0,C 180,E1 29707,E2 29707} C_VEL
LIN {X 0,Y 276.433,Z 1014.714,A -85,B 0,C 180,E1 29711.988,E2 29711.988} C_VEL
LIN {X 0,Y 246.249,Z 1049.098,A -85,B 0,C 180,E1 29715.974,E2 29715.974} C_VEL
LIN {X 0,Y 213.674,Z 1079.308,A -85,B 0,C 180,E1 29721.854,E2 29721.854} C_VEL
LIN {X 0,Y 181.766,Z 1104.084,A -85,B 0,C 180,E1 29730.531,E2 29730.531} C_VEL
LIN {X 0,Y 155.573,Z 1121.989,A -85,B 0,C 180,E1 29742.166,E2 29742.166} C_VEL
LIN {X 0,Y 137.875,Z 1134.086,A -85,B 0,C 180,E1 29756.766,E2 29756.766} C_VEL
LIN {X 0,Y 130.447,Z 1139.974,A -85,B 0,C 180,E1 29769.66,E2 29769.66} C_VEL
LIN {X 0,Y 127.885,Z 1143.235,A -85,B 0,C 180,E1 29783.21,E2 29783.21} C_VEL
LIN {X 0,Y 128.179,Z 1143.901,A -85,B 0,C 180,E1 29789.996,E2 29789.996} C_VEL
LIN {X 0,Y 128.536,Z 1143.219,A -85,B 0,C 180,E1 29803.595,E2 29803.595} C_VEL
LIN {X 0,Y 135.616,Z 1138.766,A -85,B 0,C 180,E1 29820.089,E2 29820.089} C_VEL
LIN {X 0,Y 154.62,Z 1128.309,A -85,B 0,C 180,E1 29836.855,E2 29836.855} C_VEL
LIN {X 0,Y 183.703,Z 1111.399,A -85,B 0,C 180,E1 29849.66,E2 29849.66} C_VEL
LIN {X 0,Y 217.41,Z 1088.567,A -85,B 0,C 180,E1 29858.371,E2 29858.371} C_VEL
LIN {X 0,Y 251.324,Z 1060.719,A -85,B 0,C 180,E1 29864.149,E2 29864.149} C_VEL
LIN {X 0,Y 283.175,Z 1028.646,A -85,B 0,C 180,E1 29868.045,E2 29868.045} C_VEL
LIN {X 0,Y 285.508,Z 1026.082,A -85,B 0,C 180,E1 29868.28,E2 29868.28} C_VEL
LIN {X 0,Y 287.015,Z 1020.609,A -85,B 0,C 180,E1 29872.44,E2 29872.44} C_VEL
LIN {X 0,Y 288.058,Z 1016.966,A -85,B 0,C 180,E1 29876.998,E2 29876.998} C_VEL
LIN {X 0,Y 287.955,Z 1016.544,A -85,B 0,C 180,E1 29880.005,E2 29880.005} C_VEL
LIN {X 0,Y 285.284,Z 1021.095,A -85,B 0,C 180,E1 29886.085,E2 29886.085} C_VEL
LIN {X 0,Y 281.88,Z 1027.474,A -85,B 0,C 180,E1 29890.434,E2 29890.434} C_VEL
LIN {X 0,Y 251.669,Z 1057.15,A -85,B 0,C 180,E1 29894.385,E2 29894.385} C_VEL
LIN {X 0,Y 218.358,Z 1083.781,A -85,B 0,C 180,E1 29900.247,E2 29900.247} C_VEL
LIN {X 0,Y 185.202,Z 1105.497,A -85,B 0,C 180,E1 29908.974,E2 29908.974} C_VEL
LIN {X 0,Y 155.44,Z 1121.786,A -85,B 0,C 180,E1 29922.194,E2 29922.194} C_VEL
LIN {X 0,Y 135.685,Z 1131.394,A -85,B 0,C 180,E1 29939.928,E2 29939.928} C_VEL
LIN {X 0,Y 128.548,Z 1134.702,A -85,B 0,C 180,E1 29956.406,E2 29956.406} C_VEL
LIN {X 0,Y 128.171,Z 1134.627,A -85,B 0,C 180,E1 29970.004,E2 29970.004} C_VEL
LIN {X 0,Y 131.606,Z 1131.295,A -85,B 0,C 180,E1 29986.685,E2 29986.685} C_VEL
LIN {X 0,Y 145.308,Z 1122.268,A -85,B 0,C 180,E1 30004.891,E2 30004.891} C_VEL
LIN {X 0,Y 165.698,Z 1109.423,A -85,B 0,C 180,E1 30017.821,E2 30017.821} C_VEL
LIN {X 0,Y 172.513,Z 1103.585,A -85,B 0,C 180,E1 30022.943,E2 30022.943} C_VEL
LIN {X 0,Y 180.433,Z 1097.017,A -85,B 0,C 180,E1 30027.55,E2 30027.55} C_VEL
LIN {X 0,Y 213.149,Z 1072.95,A -85,B 0,C 180,E1 30035.896,E2 30035.896} C_VEL
LIN {X 0,Y 246.557,Z 1042.918,A -85,B 0,C 180,E1 30041.7,E2 30041.7} C_VEL
LIN {X 0,Y 268.369,Z 1019.202,A -85,B 0,C 180,E1 30044.717,E2 30044.717} C_VEL
LIN {X 0,Y 271.328,Z 1012.103,A -85,B 0,C 180,E1 30049.082,E2 30049.082} C_VEL
LIN {X 0,Y 273.511,Z 1007.217,A -85,B 0,C 180,E1 30053.988,E2 30053.988} C_VEL
LIN {X 0,Y 274.605,Z 1005.483,A -85,B 0,C 180,E1 30056.841,E2 30056.841} C_VEL
LIN {X 0,Y 275.072,Z 1005.428,A -85,B 0,C 180,E1 30059.995,E2 30059.995} C_VEL
LIN {X 0,Y 273.706,Z 1011.19,A -85,B 0,C 180,E1 30066.386,E2 30066.386} C_VEL
LIN {X 0,Y 271.877,Z 1017.502,A -85,B 0,C 180,E1 30070.4,E2 30070.4} C_VEL
LIN {X 0,Y 265.696,Z 1025.296,A -85,B 0,C 180,E1 30071.352,E2 30071.352} C_VEL
LIN {X 0,Y 233.484,Z 1058.927,A -85,B 0,C 180,E1 30075.689,E2 30075.689} C_VEL
LIN {X 0,Y 198.639,Z 1088.497,A -85,B 0,C 180,E1 30082.443,E2 30082.443} C_VEL
LIN {X 0,Y 165.76,Z 1111.752,A -85,B 0,C 180,E1 30092.509,E2 30092.509} C_VEL
LIN {X 0,Y 139.124,Z 1128.589,A -85,B 0,C 180,E1 30107.242,E2 30107.242} C_VEL
LIN {X 0,Y 124.306,Z 1138.482,A -85,B 0,C 180,E1 30125.093,E2 30125.093} C_VEL
LIN {X 0,Y 119.979,Z 1142.938,A -85,B 0,C 180,E1 30142.76,E2 30142.76} C_VEL
LIN {X 0,Y 120.261,Z 1143.615,A -85,B 0,C 180,E1 30149.996,E2 30149.996} C_VEL
LIN {X 0,Y 120.755,Z 1142.947,A -85,B 0,C 180,E1 30164.49,E2 30164.49} C_VEL
LIN {X 0,Y 131.295,Z 1137.237,A -85,B 0,C 180,E1 30185.127,E2 30185.127} C_VEL
LIN {X 0,Y 156.275,Z 1124.391,A -85,B 0,C 180,E1 30202.909,E2 30202.909} C_VEL
LIN {X 0,Y 188.424,Z 1105.862,A -85,B 0,C 180,E1 30214.445,E2 30214.445} C_VEL
LIN {X 0,Y 222.56,Z 1082.362,A -85,B 0,C 180,E1 30221.899,E2 30221.899} C_VEL
LIN {X 0,Y 255.39,Z 1054.992,A -85,B 0,C 180,E1 30226.727,E2 30226.727} C_VEL
LIN {X 0,Y 280.464,Z 1029.666,A -85,B 0,C 180,E1 30229.707,E2 30229.707} C_VEL
LIN {X 0,Y 282.412,Z 1023.581,A -85,B 0,C 180,E1 30235.867,E2 30235.867} C_VEL
LIN {X 0,Y 282.59,Z 1022.469,A -85,B 0,C 180,E1 30240.005,E2 30240.005} C_VEL
LIN {X 0,Y 279.477,Z 1027.028,A -85,B 0,C 180,E1 30246.212,E2 30246.212} C_VEL
LIN {X 0,Y 277.416,Z 1030.853,A -85,B 0,C 180,E1 30249.066,E2 30249.066} C_VEL
LIN {X 0,Y 244.573,Z 1061.707,A -85,B 0,C 180,E1 30253.323,E2 30253.323} C_VEL
LIN {X 0,Y 211.545,Z 1086.709,A -85,B 0,C 180,E1 30259.016,E2 30259.016} C_VEL
LIN {X 0,Y 179.109,Z 1106.924,A -85,B 0,C 180,E1 30267.416,E2 30267.416} C_VEL
LIN {X 0,Y 150.372,Z 1121.843,A -85,B 0,C 180,E1 30279.68,E2 30279.68} C_VEL
LIN {X 0,Y 131.29,Z 1130.493,A -85,B 0,C 180,E1 30294.871,E2 30294.871} C_VEL
LIN {X 0,Y 120.779,Z 1134.982,A -85,B 0,C 180,E1 30315.513,E2 30315.513} C_VEL
LIN {X 0,Y 120.268,Z 1134.914,A -85,B 0,C 180,E1 30330.004,E2 30330.004} C_VEL
LIN {X 0,Y 124.023,Z 1131.612,A -85,B 0,C 180,E1 30347.738,E2 30347.738} C_VEL
LIN {X 0,Y 138.815,Z 1122.608,A -85,B 0,C 180,E1 30366.782,E2 30366.782} C_VEL
LIN {X 0,Y 164.038,Z 1107.566,A -85,B 0,C 180,E1 30381.542,E2 30381.542} C_VEL
LIN {X 0,Y 180.433,Z 1097.017,A -85,B 0,C 180,E1 30387.55,E2 30387.55} C_VEL
LIN {X 0,Y 189.167,Z 1089.919,A -85,B 0,C 180,E1 30391.724,E2 30391.724} C_VEL
LIN {X 0,Y 198.459,Z 1082.162,A -85,B 0,C 180,E1 30395.476,E2 30395.476} C_VEL
LIN {X 0,Y 232.661,Z 1054.269,A -85,B 0,C 180,E1 30401.789,E2 30401.789} C_VEL
LIN {X 0,Y 262.543,Z 1024.115,A -85,B 0,C 180,E1 30405.775,E2 30405.775} C_VEL
LIN {X 0,Y 264.2,Z 1021.638,A -85,B 0,C 180,E1 30406.772,E2 30406.772} C_VEL
LIN {X 0,Y 267.198,Z 1015.099,A -85,B 0,C 180,E1 30411.868,E2 30411.868} C_VEL
LIN {X 0,Y 269.397,Z 1011.626,A -85,B 0,C 180,E1 30416.78,E2 30416.78} C_VEL
LIN {X 0,Y 269.95,Z 1011.52,A -85,B 0,C 180,E1 30419.995,E2 30419.995} C_VEL
LIN {X 0,Y 268.16,Z 1017.344,A -85,B 0,C 180,E1 30426.465,E2 30426.465} C_VEL
LIN {X 0,Y 266.261,Z 1022.376,A -85,B 0,C 180,E1 30429.395,E2 30429.395} C_VEL
LIN {X 0,Y 235.922,Z 1054.171,A -85,B 0,C 180,E1 30433.114,E2 30433.114} C_VEL
LIN {X 0,Y 204.911,Z 1080.944,A -85,B 0,C 180,E1 30438.286,E2 30438.286} C_VEL
LIN {X 0,Y 172.349,Z 1104.411,A -85,B 0,C 180,E1 30446.358,E2 30446.358} C_VEL
LIN {X 0,Y 141.568,Z 1123.359,A -85,B 0,C 180,E1 30459.297,E2 30459.297} C_VEL
LIN {X 0,Y 121.707,Z 1135.071,A -85,B 0,C 180,E1 30476.028,E2 30476.028} C_VEL
LIN {X 0,Y 113.021,Z 1141.309,A -85,B 0,C 180,E1 30494.486,E2 30494.486} C_VEL
LIN {X 0,Y 112.34,Z 1143.329,A -85,B 0,C 180,E1 30509.996,E2 30509.996} C_VEL
LIN {X 0,Y 113.007,Z 1142.675,A -85,B 0,C 180,E1 30525.507,E2 30525.507} C_VEL
LIN {X 0,Y 124.739,Z 1136.983,A -85,B 0,C 180,E1 30547.275,E2 30547.275} C_VEL
LIN {X 0,Y 151.481,Z 1124.162,A -85,B 0,C 180,E1 30565.379,E2 30565.379} C_VEL
LIN {X 0,Y 185.045,Z 1105.666,A -85,B 0,C 180,E1 30576.728,E2 30576.728} C_VEL
LIN {X 0,Y 220.169,Z 1082.204,A -85,B 0,C 180,E1 30583.911,E2 30583.911} C_VEL
LIN {X 0,Y 252.611,Z 1055.845,A -85,B 0,C 180,E1 30588.381,E2 30588.381} C_VEL
LIN {X 0,Y 274.003,Z 1035.259,A -85,B 0,C 180,E1 30590.678,E2 30590.678} C_VEL
LIN {X 0,Y 275.301,Z 1033.613,A -85,B 0,C 180,E1 30591.104,E2 30591.104} C_VEL
LIN {X 0,Y 277.084,Z 1028.608,A -85,B 0,C 180,E1 30596.879,E2 30596.879} C_VEL
LIN {X 0,Y 276.984,Z 1028.157,A -85,B 0,C 180,E1 30600.005,E2 30600.005} C_VEL
LIN {X 0,Y 273.631,Z 1032.956,A -85,B 0,C 180,E1 30606.278,E2 30606.278} C_VEL
LIN {X 0,Y 271.535,Z 1035.75,A -85,B 0,C 180,E1 30607.991,E2 30607.991} C_VEL
LIN {X 0,Y 237.68,Z 1066.07,A -85,B 0,C 180,E1 30612.187,E2 30612.187} C_VEL
LIN {X 0,Y 202.765,Z 1091.041,A -85,B 0,C 180,E1 30618.167,E2 30618.167} C_VEL
LIN {X 0,Y 169.478,Z 1110.269,A -85,B 0,C 180,E1 30626.929,E2 30626.929} C_VEL
LIN {X 0,Y 139.693,Z 1124.488,A -85,B 0,C 180,E1 30640.473,E2 30640.473} C_VEL
LIN {X 0,Y 121.921,Z 1131.901,A -85,B 0,C 180,E1 30656.106,E2 30656.106} C_VEL
LIN {X 0,Y 113.042,Z 1135.262,A -85,B 0,C 180,E1 30674.498,E2 30674.498} C_VEL
LIN {X 0,Y 112.345,Z 1135.2,A -85,B 0,C 180,E1 30690.004,E2 30690.004} C_VEL
LIN {X 0,Y 116.484,Z 1131.929,A -85,B 0,C 180,E1 30708.929,E2 30708.929} C_VEL
LIN {X 0,Y 132.5,Z 1122.947,A -85,B 0,C 180,E1 30728.852,E2 30728.852} C_VEL
LIN {X 0,Y 156.625,Z 1109.427,A -85,B 0,C 180,E1 30742.751,E2 30742.751} C_VEL
LIN {X 0,Y 186.98,Z 1090.287,A -85,B 0,C 180,E1 30752.751,E2 30752.751} C_VEL
LIN {X 0,Y 198.459,Z 1082.162,A -85,B 0,C 180,E1 30755.476,E2 30755.476} C_VEL
LIN {X 0,Y 208.204,Z 1073.886,A -85,B 0,C 180,E1 30758.826,E2 30758.826} C_VEL
LIN {X 0,Y 218.374,Z 1064.923,A -85,B 0,C 180,E1 30761.848,E2 30761.848} C_VEL
LIN {X 0,Y 251.939,Z 1033.983,A -85,B 0,C 180,E1 30766.485,E2 30766.485} C_VEL
LIN {X 0,Y 257.474,Z 1028.101,A -85,B 0,C 180,E1 30767.12,E2 30767.12} C_VEL
LIN {X 0,Y 259.248,Z 1025.738,A -85,B 0,C 180,E1 30767.944,E2 30767.944} C_VEL
LIN {X 0,Y 262.681,Z 1019.434,A -85,B 0,C 180,E1 30773.852,E2 30773.852} C_VEL
LIN {X 0,Y 264.017,Z 1017.603,A -85,B 0,C 180,E1 30776.714,E2 30776.714} C_VEL
LIN {X 0,Y 264.602,Z 1017.452,A -85,B 0,C 180,E1 30779.995,E2 30779.995} C_VEL
LIN {X 0,Y 262.589,Z 1023.557,A -85,B 0,C 180,E1 30786.603,E2 30786.603} C_VEL
LIN {X 0,Y 261.352,Z 1026.059,A -85,B 0,C 180,E1 30788.039,E2 30788.039} C_VEL
LIN {X 0,Y 227.883,Z 1059.538,A -85,B 0,C 180,E1 30792.008,E2 30792.008} C_VEL
LIN {X 0,Y 192.676,Z 1087.887,A -85,B 0,C 180,E1 30798.015,E2 30798.015} C_VEL
LIN {X 0,Y 157.553,Z 1110.977,A -85,B 0,C 180,E1 30807.473,E2 30807.473} C_VEL
LIN {X 0,Y 127.5,Z 1127.925,A -85,B 0,C 180,E1 30822.295,E2 30822.295} C_VEL
LIN {X 0,Y 109.985,Z 1137.748,A -85,B 0,C 180,E1 30841.253,E2 30841.253} C_VEL
LIN {X 0,Y 104.203,Z 1142.344,A -85,B 0,C 180,E1 30861.657,E2 30861.657} C_VEL
LIN {X 0,Y 104.445,Z 1143.043,A -85,B 0,C 180,E1 30869.995,E2 30869.995} C_VEL
LIN {X 0,Y 105.324,Z 1142.405,A -85,B 0,C 180,E1 30886.67,E2 30886.67} C_VEL
LIN {X 0,Y 118.359,Z 1136.726,A -85,B 0,C 180,E1 30909.664,E2 30909.664} C_VEL
LIN {X 0,Y 144.367,Z 1125.111,A -85,B 0,C 180,E1 30926.857,E2 30926.857} C_VEL
LIN {X 0,Y 176.539,Z 1108.547,A -85,B 0,C 180,E1 30937.753,E2 30937.753} C_VEL
LIN {X 0,Y 211.3,Z 1086.894,A -85,B 0,C 180,E1 30944.885,E2 30944.885} C_VEL
LIN {X 0,Y 247.574,Z 1058.873,A -85,B 0,C 180,E1 30949.795,E2 30949.795} C_VEL
LIN {X 0,Y 268.03,Z 1039.871,A -85,B 0,C 180,E1 30951.919,E2 30951.919} C_VEL
LIN {X 0,Y 269.905,Z 1037.898,A -85,B 0,C 180,E1 30952.312,E2 30952.312} C_VEL
LIN {X 0,Y 271.456,Z 1034.326,A -85,B 0,C 180,E1 30956.814,E2 30956.814} C_VEL
LIN {X 0,Y 271.366,Z 1033.854,A -85,B 0,C 180,E1 30960.005,E2 30960.005} C_VEL
LIN {X 0,Y 268.425,Z 1037.336,A -85,B 0,C 180,E1 30965.125,E2 30965.125} C_VEL
LIN {X 0,Y 266.712,Z 1039.521,A -85,B 0,C 180,E1 30966.662,E2 30966.662} C_VEL
LIN {X 0,Y 234.346,Z 1067.523,A -85,B 0,C 180,E1 30970.483,E2 30970.483} C_VEL
LIN {X 0,Y 198.724,Z 1092.253,A -85,B 0,C 180,E1 30976.267,E2 30976.267} C_VEL
LIN {X 0,Y 162.996,Z 1111.977,A -85,B 0,C 180,E1 30985.331,E2 30985.331} C_VEL
LIN {X 0,Y 134.218,Z 1124.846,A -85,B 0,C 180,E1 30997.998,E2 30997.998} C_VEL
LIN {X 0,Y 115.253,Z 1132.155,A -85,B 0,C 180,E1 31013.848,E2 31013.848} C_VEL
LIN {X 0,Y 105.364,Z 1135.542,A -85,B 0,C 180,E1 31033.336,E2 31033.336} C_VEL
LIN {X 0,Y 104.431,Z 1135.487,A -85,B 0,C 180,E1 31050.005,E2 31050.005} C_VEL
LIN {X 0,Y 109.018,Z 1132.245,A -85,B 0,C 180,E1 31070.28,E2 31070.28} C_VEL
LIN {X 0,Y 126.38,Z 1123.286,A -85,B 0,C 180,E1 31091.124,E2 31091.124} C_VEL
LIN {X 0,Y 154.599,Z 1108.309,A -85,B 0,C 180,E1 31106.189,E2 31106.189} C_VEL
LIN {X 0,Y 187.179,Z 1088.135,A -85,B 0,C 180,E1 31115.849,E2 31115.849} C_VEL
LIN {X 0,Y 218.374,Z 1064.923,A -85,B 0,C 180,E1 31121.848,E2 31121.848} C_VEL
LIN {X 0,Y 228.694,Z 1055.441,A -85,B 0,C 180,E1 31124.557,E2 31124.557} C_VEL
LIN {X 0,Y 239.048,Z 1045.327,A -85,B 0,C 180,E1 31126.983,E2 31126.983} C_VEL
LIN {X 0,Y 253.12,Z 1031.485,A -85,B 0,C 180,E1 31128.57,E2 31128.57} C_VEL
LIN {X 0,Y 254.715,Z 1029.207,A -85,B 0,C 180,E1 31129.745,E2 31129.745} C_VEL
LIN {X 0,Y 257.823,Z 1024.347,A -85,B 0,C 180,E1 31135.142,E2 31135.142} C_VEL
LIN {X 0,Y 259.212,Z 1023.36,A -85,B 0,C 180,E1 31139.995,E2 31139.995} C_VEL
LIN {X 0,Y 257.019,Z 1028.818,A -85,B 0,C 180,E1 31146.194,E2 31146.194} C_VEL
LIN {X 0,Y 254.647,Z 1031.674,A -85,B 0,C 180,E1 31146.81,E2 31146.81} C_VEL
LIN {X 0,Y 222.811,Z 1062.055,A -85,B 0,C 180,E1 31150.446,E2 31150.446} C_VEL
LIN {X 0,Y 188.64,Z 1088.609,A -85,B 0,C 180,E1 31155.99,E2 31155.99} C_VEL
LIN {X 0,Y 153.948,Z 1110.59,A -85,B 0,C 180,E1 31164.769,E2 31164.769} C_VEL
LIN {X 0,Y 123.28,Z 1126.977,A -85,B 0,C 180,E1 31178.709,E2 31178.709} C_VEL
LIN {X 0,Y 102.964,Z 1137.427,A -85,B 0,C 180,E1 31199.086,E2 31199.086} C_VEL
LIN {X 0,Y 96.315,Z 1142.046,A -85,B 0,C 180,E1 31220.968,E2 31220.968} C_VEL
LIN {X 0,Y 96.519,Z 1142.756,A -85,B 0,C 180,E1 31229.995,E2 31229.995} C_VEL
LIN {X 0,Y 97.657,Z 1142.133,A -85,B 0,C 180,E1 31248.022,E2 31248.022} C_VEL
LIN {X 0,Y 112.219,Z 1136.469,A -85,B 0,C 180,E1 31272.315,E2 31272.315} C_VEL
LIN {X 0,Y 140.054,Z 1124.882,A -85,B 0,C 180,E1 31289.665,E2 31289.665} C_VEL
LIN {X 0,Y 173.901,Z 1108.196,A -85,B 0,C 180,E1 31300.308,E2 31300.308} C_VEL
LIN {X 0,Y 209.953,Z 1086.291,A -85,B 0,C 180,E1 31307.141,E2 31307.141} C_VEL
LIN {X 0,Y 248.062,Z 1057.23,A -85,B 0,C 180,E1 31311.832,E2 31311.832} C_VEL
LIN {X 0,Y 264.418,Z 1042.269,A -85,B 0,C 180,E1 31313.443,E2 31313.443} C_VEL
LIN {X 0,Y 265.583,Z 1039.81,A -85,B 0,C 180,E1 31316.744,E2 31316.744} C_VEL
LIN {X 0,Y 265.485,Z 1039.332,A -85,B 0,C 180,E1 31320.005,E2 31320.005} C_VEL
LIN {X 0,Y 262.528,Z 1042.741,A -85,B 0,C 180,E1 31324.986,E2 31324.986} C_VEL
LIN {X 0,Y 258.146,Z 1046.825,A -85,B 0,C 180,E1 31325.68,E2 31325.68} C_VEL
LIN {X 0,Y 221.728,Z 1075.968,A -85,B 0,C 180,E1 31329.962,E2 31329.962} C_VEL
LIN {X 0,Y 185.655,Z 1098.756,A -85,B 0,C 180,E1 31336.146,E2 31336.146} C_VEL
LIN {X 0,Y 150.763,Z 1116.205,A -85,B 0,C 180,E1 31345.576,E2 31345.576} C_VEL
LIN {X 0,Y 123.455,Z 1127.366,A -85,B 0,C 180,E1 31358.714,E2 31358.714} C_VEL
LIN {X 0,Y 105.767,Z 1133.385,A -85,B 0,C 180,E1 31375.152,E2 31375.152} C_VEL
LIN {X 0,Y 97.708,Z 1135.822,A -85,B 0,C 180,E1 31391.988,E2 31391.988} C_VEL
LIN {X 0,Y 96.505,Z 1135.774,A -85,B 0,C 180,E1 31410.005,E2 31410.005} C_VEL
LIN {X 0,Y 99.843,Z 1133.442,A -85,B 0,C 180,E1 31427.625,E2 31427.625} C_VEL
LIN {X 0,Y 112.965,Z 1127.148,A -85,B 0,C 180,E1 31447.355,E2 31447.355} C_VEL
LIN {X 0,Y 139.441,Z 1114.37,A -85,B 0,C 180,E1 31464.373,E2 31464.373} C_VEL
LIN {X 0,Y 170.886,Z 1096.882,A -85,B 0,C 180,E1 31475.017,E2 31475.017} C_VEL
LIN {X 0,Y 204.532,Z 1074.256,A -85,B 0,C 180,E1 31482.038,E2 31482.038} C_VEL
LIN {X 0,Y 239.048,Z 1045.327,A -85,B 0,C 180,E1 31486.983,E2 31486.983} C_VEL
LIN {X 0,Y 245.991,Z 1038.25,A -85,B 0,C 180,E1 31488.635,E2 31488.635} C_VEL
LIN {X 0,Y 249.793,Z 1033.507,A -85,B 0,C 180,E1 31491.084,E2 31491.084} C_VEL
LIN {X 0,Y 252.924,Z 1029.247,A -85,B 0,C 180,E1 31496.57,E2 31496.57} C_VEL
LIN {X 0,Y 253.59,Z 1029.053,A -85,B 0,C 180,E1 31499.995,E2 31499.995} C_VEL
LIN {X 0,Y 251.772,Z 1033.21,A -85,B 0,C 180,E1 31504.978,E2 31504.978} C_VEL
LIN {X 0,Y 221.22,Z 1061.815,A -85,B 0,C 180,E1 31508.401,E2 31508.401} C_VEL
LIN {X 0,Y 186.554,Z 1088.197,A -85,B 0,C 180,E1 31513.576,E2 31513.576} C_VEL
LIN {X 0,Y 150.703,Z 1110.204,A -85,B 0,C 180,E1 31521.942,E2 31521.942} C_VEL
LIN {X 0,Y 118.011,Z 1126.775,A -85,B 0,C 180,E1 31535.801,E2 31535.801} C_VEL
LIN {X 0,Y 96.088,Z 1137.105,A -85,B 0,C 180,E1 31556.598,E2 31556.598} C_VEL
LIN {X 0,Y 88.44,Z 1141.748,A -85,B 0,C 180,E1 31580.156,E2 31580.156} C_VEL
LIN {X 0,Y 88.62,Z 1142.471,A -85,B 0,C 180,E1 31589.994,E2 31589.994} C_VEL
LIN {X 0,Y 90.055,Z 1141.861,A -85,B 0,C 180,E1 31609.603,E2 31609.603} C_VEL
LIN {X 0,Y 106.354,Z 1136.213,A -85,B 0,C 180,E1 31635.262,E2 31635.262} C_VEL
LIN {X 0,Y 136.095,Z 1124.654,A -85,B 0,C 180,E1 31652.648,E2 31652.648} C_VEL
LIN {X 0,Y 171.556,Z 1107.871,A -85,B 0,C 180,E1 31662.946,E2 31662.946} C_VEL
LIN {X 0,Y 208.991,Z 1085.656,A -85,B 0,C 180,E1 31669.415,E2 31669.415} C_VEL
LIN {X 0,Y 247.046,Z 1057.12,A -85,B 0,C 180,E1 31673.681,E2 31673.681} C_VEL
LIN {X 0,Y 257.995,Z 1047.487,A -85,B 0,C 180,E1 31674.669,E2 31674.669} C_VEL
LIN {X 0,Y 259.69,Z 1045.28,A -85,B 0,C 180,E1 31676.67,E2 31676.67} C_VEL
LIN {X 0,Y 259.579,Z 1044.805,A -85,B 0,C 180,E1 31680.005,E2 31680.005} C_VEL
LIN {X 0,Y 257.394,Z 1046.947,A -85,B 0,C 180,E1 31683.624,E2 31683.624} C_VEL
LIN {X 0,Y 250.123,Z 1053.291,A -85,B 0,C 180,E1 31684.582,E2 31684.582} C_VEL
LIN {X 0,Y 215.623,Z 1079.357,A -85,B 0,C 180,E1 31688.516,E2 31688.516} C_VEL
LIN {X 0,Y 181.357,Z 1100.179,A -85,B 0,C 180,E1 31694.13,E2 31694.13} C_VEL
LIN {X 0,Y 142.54,Z 1118.548,A -85,B 0,C 180,E1 31704.376,E2 31704.376} C_VEL
LIN {X 0,Y 110.438,Z 1130.246,A -85,B 0,C 180,E1 31721.195,E2 31721.195} C_VEL
LIN {X 0,Y 93.749,Z 1135.176,A -85,B 0,C 180,E1 31741.088,E2 31741.088} C_VEL
LIN {X 0,Y 88.422,Z 1136.384,A -85,B 0,C 180,E1 31760.166,E2 31760.166} C_VEL
LIN {X 0,Y 88.577,Z 1136.06,A -85,B 0,C 180,E1 31770.006,E2 31770.006} C_VEL
LIN {X 0,Y 92.326,Z 1133.748,A -85,B 0,C 180,E1 31789.113,E2 31789.113} C_VEL
LIN {X 0,Y 106.449,Z 1127.583,A -85,B 0,C 180,E1 31809.708,E2 31809.708} C_VEL
LIN {X 0,Y 134.937,Z 1114.73,A -85,B 0,C 180,E1 31827.136,E2 31827.136} C_VEL
LIN {X 0,Y 167.659,Z 1097.278,A -85,B 0,C 180,E1 31837.5,E2 31837.5} C_VEL
LIN {X 0,Y 203.912,Z 1073.39,A -85,B 0,C 180,E1 31844.454,E2 31844.454} C_VEL
LIN {X 0,Y 239.382,Z 1043.964,A -85,B 0,C 180,E1 31849.08,E2 31849.08} C_VEL
LIN {X 0,Y 249.253,Z 1034.309,A -85,B 0,C 180,E1 31850.338,E2 31850.338} C_VEL
LIN {X 0,Y 249.793,Z 1033.507,A -85,B 0,C 180,E1 31851.084,E2 31851.084} C_VEL
LIN {X 0,Y 249.731,Z 1032.749,A -85,B 0,C 180,E1 31854.086,E2 31854.086} C_VEL
LIN {X 0,Y 247.73,Z 1034.778,A -85,B 0,C 180,E1 31859.248,E2 31859.248} C_VEL
LIN {X 0,Y 246.56,Z 1037.367,A -85,B 0,C 180,E1 31863.508,E2 31863.508} C_VEL
LIN {X 0,Y 229.557,Z 1053.338,A -85,B 0,C 180,E1 31865.334,E2 31865.334} C_VEL
LIN {X 0,Y 195.339,Z 1080.473,A -85,B 0,C 180,E1 31869.474,E2 31869.474} C_VEL
LIN {X 0,Y 157.597,Z 1104.466,A -85,B 0,C 180,E1 31876.485,E2 31876.485} C_VEL
LIN {X 0,Y 120.642,Z 1123.252,A -85,B 0,C 180,E1 31888.734,E2 31888.734} C_VEL
LIN {X 0,Y 92.691,Z 1135.373,A -85,B 0,C 180,E1 31909.293,E2 31909.293} C_VEL
LIN {X 0,Y 82.556,Z 1140.074,A -85,B 0,C 180,E1 31928.519,E2 31928.519} C_VEL
LIN {X 0,Y 80.687,Z 1142.184,A -85,B 0,C 180,E1 31949.994,E2 31949.994} C_VEL
LIN {X 0,Y 84.029,Z 1141.088,A -85,B 0,C 180,E1 31976.009,E2 31976.009} C_VEL
LIN {X 0,Y 100.775,Z 1135.956,A -85,B 0,C 180,E1 31998.56,E2 31998.56} C_VEL
LIN {X 0,Y 132.531,Z 1124.426,A -85,B 0,C 180,E1 32015.795,E2 32015.795} C_VEL
LIN {X 0,Y 167.812,Z 1108.473,A -85,B 0,C 180,E1 32025.282,E2 32025.282} C_VEL
LIN {X 0,Y 206.681,Z 1086.157,A -85,B 0,C 180,E1 32031.502,E2 32031.502} C_VEL
LIN {X 0,Y 245.372,Z 1057.757,A -85,B 0,C 180,E1 32035.476,E2 32035.476} C_VEL
LIN {X 0,Y 251.627,Z 1052.364,A -85,B 0,C 180,E1 32035.993,E2 32035.993} C_VEL
LIN {X 0,Y 253.577,Z 1050.539,A -85,B 0,C 180,E1 32036.589,E2 32036.589} C_VEL
LIN {X 0,Y 253.475,Z 1050.042,A -85,B 0,C 180,E1 32040.005,E2 32040.005} C_VEL
LIN {X 0,Y 251.979,Z 1051.352,A -85,B 0,C 180,E1 32042.358,E2 32042.358} C_VEL
LIN {X 0,Y 217.825,Z 1077.37,A -85,B 0,C 180,E1 32045.963,E2 32045.963} C_VEL
LIN {X 0,Y 178.487,Z 1100.896,A -85,B 0,C 180,E1 32051.774,E2 32051.774} C_VEL
LIN {X 0,Y 139.791,Z 1118.576,A -85,B 0,C 180,E1 32061.15,E2 32061.15} C_VEL
LIN {X 0,Y 105.253,Z 1130.491,A -85,B 0,C 180,E1 32077.857,E2 32077.857} C_VEL
LIN {X 0,Y 86.774,Z 1135.448,A -85,B 0,C 180,E1 32098.511,E2 32098.511} C_VEL
LIN {X 0,Y 80.574,Z 1136.662,A -85,B 0,C 180,E1 32119.197,E2 32119.197} C_VEL
LIN {X 0,Y 80.646,Z 1136.347,A -85,B 0,C 180,E1 32130.006,E2 32130.006} C_VEL
LIN {X 0,Y 84.866,Z 1134.054,A -85,B 0,C 180,E1 32150.868,E2 32150.868} C_VEL
LIN {X 0,Y 100.441,Z 1127.911,A -85,B 0,C 180,E1 32172.617,E2 32172.617} C_VEL
LIN {X 0,Y 130.752,Z 1115.093,A -85,B 0,C 180,E1 32190.094,E2 32190.094} C_VEL
LIN {X 0,Y 164.767,Z 1097.671,A -85,B 0,C 180,E1 32200.068,E2 32200.068} C_VEL
LIN {X 0,Y 201.926,Z 1073.821,A -85,B 0,C 180,E1 32206.629,E2 32206.629} C_VEL
LIN {X 0,Y 238.007,Z 1044.44,A -85,B 0,C 180,E1 32210.955,E2 32210.955} C_VEL
LIN {X 0,Y 244.293,Z 1038.361,A -85,B 0,C 180,E1 32211.783,E2 32211.783} C_VEL
LIN {X 0,Y 247.199,Z 1034.973,A -85,B 0,C 180,E1 32216.491,E2 32216.491} C_VEL
LIN {X 0,Y 247.73,Z 1034.778,A -85,B 0,C 180,E1 32219.248,E2 32219.248} C_VEL
LIN {X 0,Y 245.942,Z 1036.888,A -85,B 0,C 180,E1 32220.795,E2 32220.795} C_VEL
LIN {X 0,Y 238.246,Z 1044.576,A -85,B 0,C 180,E1 32222.416,E2 32222.416} C_VEL
LIN {X 0,Y 234.692,Z 1047.825,A -85,B 0,C 180,E1 32222.784,E2 32222.784} C_VEL
LIN {X 0,Y 197.769,Z 1077.569,A -85,B 0,C 180,E1 32226.616,E2 32226.616} C_VEL
LIN {X 0,Y 158.87,Z 1102.161,A -85,B 0,C 180,E1 32232.84,E2 32232.84} C_VEL
LIN {X 0,Y 122.941,Z 1120.151,A -85,B 0,C 180,E1 32242.791,E2 32242.791} C_VEL
LIN {X 0,Y 95.401,Z 1131.688,A -85,B 0,C 180,E1 32257.621,E2 32257.621} C_VEL
LIN {X 0,Y 77.008,Z 1138.935,A -85,B 0,C 180,E1 32281.161,E2 32281.161} C_VEL
LIN {X 0,Y 72.768,Z 1141.897,A -85,B 0,C 180,E1 32309.993,E2 32309.993} C_VEL
LIN {X 0,Y 75.123,Z 1141.317,A -85,B 0,C 180,E1 32333.715,E2 32333.715} C_VEL
LIN {X 0,Y 95.573,Z 1135.698,A -85,B 0,C 180,E1 32362.228,E2 32362.228} C_VEL
LIN {X 0,Y 129.394,Z 1124.199,A -85,B 0,C 180,E1 32379.099,E2 32379.099} C_VEL
LIN {X 0,Y 166.046,Z 1108.22,A -85,B 0,C 180,E1 32388.029,E2 32388.029} C_VEL
LIN {X 0,Y 205.636,Z 1086.001,A -85,B 0,C 180,E1 32393.745,E2 32393.745} C_VEL
LIN {X 0,Y 245.369,Z 1057.236,A -85,B 0,C 180,E1 32397.395,E2 32397.395} C_VEL
LIN {X 0,Y 247.408,Z 1055.435,A -85,B 0,C 180,E1 32397.913,E2 32397.913} C_VEL
LIN {X 0,Y 246.827,Z 1055.643,A -85,B 0,C 180,E1 32400.732,E2 32400.732} C_VEL
LIN {X 0,Y 241.849,Z 1059.552,A -85,B 0,C 180,E1 32401.488,E2 32401.488} C_VEL
LIN {X 0,Y 204.842,Z 1085.441,A -85,B 0,C 180,E1 32405.226,E2 32405.226} C_VEL
LIN {X 0,Y 165.599,Z 1106.649,A -85,B 0,C 180,E1 32411.218,E2 32411.218} C_VEL
LIN {X 0,Y 125.779,Z 1122.856,A -85,B 0,C 180,E1 32421.698,E2 32421.698} C_VEL
LIN {X 0,Y 95.554,Z 1132.022,A -85,B 0,C 180,E1 32437.757,E2 32437.757} C_VEL
LIN {X 0,Y 75.22,Z 1136.656,A -85,B 0,C 180,E1 32466.317,E2 32466.317} C_VEL
LIN {X 0,Y 72.713,Z 1136.634,A -85,B 0,C 180,E1 32490.007,E2 32490.007} C_VEL
LIN {X 0,Y 77.498,Z 1134.361,A -85,B 0,C 180,E1 32512.96,E2 32512.96} C_VEL
LIN {X 0,Y 94.711,Z 1128.24,A -85,B 0,C 180,E1 32535.894,E2 32535.894} C_VEL
LIN {X 0,Y 126.952,Z 1115.453,A -85,B 0,C 180,E1 32553.226,E2 32553.226} C_VEL
LIN {X 0,Y 162.216,Z 1098.064,A -85,B 0,C 180,E1 32562.723,E2 32562.723} C_VEL
LIN {X 0,Y 200.232,Z 1074.253,A -85,B 0,C 180,E1 32568.85,E2 32568.85} C_VEL
LIN {X 0,Y 237.625,Z 1044.219,A -85,B 0,C 180,E1 32572.929,E2 32572.929} C_VEL
LIN {X 0,Y 239.595,Z 1042.232,A -85,B 0,C 180,E1 32573.761,E2 32573.761} C_VEL
LIN {X 0,Y 241.206,Z 1040.525,A -85,B 0,C 180,E1 32576.403,E2 32576.403} C_VEL
LIN {X 0,Y 241.803,Z 1040.632,A -85,B 0,C 180,E1 32580.7,E2 32580.7} C_VEL
LIN {X 0,Y 240.49,Z 1042.401,A -85,B 0,C 180,E1 32582.281,E2 32582.281} C_VEL
LIN {X 0,Y 234.692,Z 1047.825,A -85,B 0,C 180,E1 32582.784,E2 32582.784} C_VEL
LIN {X 0,Y 221.192,Z 1059.06,A -85,B 0,C 180,E1 32582.916,E2 32582.916} C_VEL
LIN {X 0,Y 207.263,Z 1069.614,A -85,B 0,C 180,E1 32583.15,E2 32583.15} C_VEL
LIN {X 0,Y 167.914,Z 1095.771,A -85,B 0,C 180,E1 32588.121,E2 32588.121} C_VEL
LIN {X 0,Y 126.49,Z 1117.023,A -85,B 0,C 180,E1 32597.102,E2 32597.102} C_VEL
LIN {X 0,Y 90.641,Z 1131.343,A -85,B 0,C 180,E1 32613.523,E2 32613.523} C_VEL
LIN {X 0,Y 68.448,Z 1139.223,A -85,B 0,C 180,E1 32641.955,E2 32641.955} C_VEL
LIN {X 0,Y 64.829,Z 1141.61,A -85,B 0,C 180,E1 32669.992,E2 32669.992} C_VEL
LIN {X 0,Y 68.261,Z 1140.926,A -85,B 0,C 180,E1 32697.749,E2 32697.749} C_VEL
LIN {X 0,Y 90.804,Z 1135.442,A -85,B 0,C 180,E1 32726.302,E2 32726.302} C_VEL
LIN {X 0,Y 126.707,Z 1123.972,A -85,B 0,C 180,E1 32742.555,E2 32742.555} C_VEL
LIN {X 0,Y 164.551,Z 1108.027,A -85,B 0,C 180,E1 32750.802,E2 32750.802} C_VEL
LIN {X 0,Y 203.419,Z 1086.759,A -85,B 0,C 180,E1 32755.855,E2 32755.855} C_VEL
LIN {X 0,Y 241.143,Z 1060.202,A -85,B 0,C 180,E1 32759.171,E2 32759.171} C_VEL
LIN {X 0,Y 238.1,Z 1062.487,A -85,B 0,C 180,E1 32759.844,E2 32759.844} C_VEL
LIN {X 0,Y 200.558,Z 1087.75,A -85,B 0,C 180,E1 32763.364,E2 32763.364} C_VEL
LIN {X 0,Y 160.65,Z 1108.479,A -85,B 0,C 180,E1 32769.034,E2 32769.034} C_VEL
LIN {X 0,Y 119.393,Z 1124.326,A -85,B 0,C 180,E1 32779.379,E2 32779.379} C_VEL
LIN {X 0,Y 85.96,Z 1133.394,A -85,B 0,C 180,E1 32797.479,E2 32797.479} C_VEL
LIN {X 0,Y 67.932,Z 1136.932,A -85,B 0,C 180,E1 32823.592,E2 32823.592} C_VEL
LIN {X 0,Y 64.777,Z 1136.922,A -85,B 0,C 180,E1 32850.008,E2 32850.008} C_VEL
LIN {X 0,Y 70.256,Z 1134.668,A -85,B 0,C 180,E1 32875.486,E2 32875.486} C_VEL
LIN {X 0,Y 89.351,Z 1128.567,A -85,B 0,C 180,E1 32899.565,E2 32899.565} C_VEL
LIN {X 0,Y 123.556,Z 1115.812,A -85,B 0,C 180,E1 32916.539,E2 32916.539} C_VEL
LIN {X 0,Y 159.97,Z 1098.486,A -85,B 0,C 180,E1 32925.452,E2 32925.452} C_VEL
LIN {X 0,Y 198.844,Z 1074.684,A -85,B 0,C 180,E1 32931.104,E2 32931.104} C_VEL
LIN {X 0,Y 232.496,Z 1048.407,A -85,B 0,C 180,E1 32934.482,E2 32934.482} C_VEL
LIN {X 0,Y 234.505,Z 1046.65,A -85,B 0,C 180,E1 32935.278,E2 32935.278} C_VEL
LIN {X 0,Y 236.016,Z 1045.908,A -85,B 0,C 180,E1 32940.452,E2 32940.452} C_VEL
LIN {X 0,Y 216.392,Z 1062.517,A -85,B 0,C 180,E1 32942.278,E2 32942.278} C_VEL
LIN {X 0,Y 207.263,Z 1069.614,A -85,B 0,C 180,E1 32943.15,E2 32943.15} C_VEL
LIN {X 0,Y 192.779,Z 1079.561,A -85,B 0,C 180,E1 32943.459,E2 32943.459} C_VEL
LIN {X 0,Y 179.757,Z 1087.706,A -85,B 0,C 180,E1 32943.706,E2 32943.706} C_VEL
LIN {X 0,Y 177.961,Z 1088.77,A -85,B 0,C 180,E1 32943.905,E2 32943.905} C_VEL
LIN {X 0,Y 138.213,Z 1110.376,A -85,B 0,C 180,E1 32950.247,E2 32950.247} C_VEL
LIN {X 0,Y 98.19,Z 1126.938,A -85,B 0,C 180,E1 32962.562,E2 32962.562} C_VEL
LIN {X 0,Y 67.151,Z 1137.089,A -85,B 0,C 180,E1 32987.529,E2 32987.529} C_VEL
LIN {X 0,Y 57.226,Z 1140.556,A -85,B 0,C 180,E1 33014.68,E2 33014.68} C_VEL
LIN {X 0,Y 56.886,Z 1141.323,A -85,B 0,C 180,E1 33029.991,E2 33029.991} C_VEL
LIN {X 0,Y 60.736,Z 1140.772,A -85,B 0,C 180,E1 33059.832,E2 33059.832} C_VEL
LIN {X 0,Y 86.547,Z 1135.185,A -85,B 0,C 180,E1 33090.797,E2 33090.797} C_VEL
LIN {X 0,Y 124.5,Z 1123.745,A -85,B 0,C 180,E1 33106.149,E2 33106.149} C_VEL
LIN {X 0,Y 163.445,Z 1107.834,A -85,B 0,C 180,E1 33113.628,E2 33113.628} C_VEL
LIN {X 0,Y 204.107,Z 1085.935,A -85,B 0,C 180,E1 33118.232,E2 33118.232} C_VEL
LIN {X 0,Y 218.045,Z 1076.954,A -85,B 0,C 180,E1 33119.427,E2 33119.427} C_VEL
LIN {X 0,Y 177.877,Z 1100.057,A -85,B 0,C 180,E1 33123.494,E2 33123.494} C_VEL
LIN {X 0,Y 138.111,Z 1117.279,A -85,B 0,C 180,E1 33130.052,E2 33130.052} C_VEL
LIN {X 0,Y 104.508,Z 1128.126,A -85,B 0,C 180,E1 33139.988,E2 33139.988} C_VEL
LIN {X 0,Y 76.051,Z 1134.708,A -85,B 0,C 180,E1 33157.376,E2 33157.376} C_VEL
LIN {X 0,Y 60.851,Z 1137.205,A -85,B 0,C 180,E1 33180.23,E2 33180.23} C_VEL
LIN {X 0,Y 56.839,Z 1137.209,A -85,B 0,C 180,E1 33210.009,E2 33210.009} C_VEL
LIN {X 0,Y 63.198,Z 1134.974,A -85,B 0,C 180,E1 33238.578,E2 33238.578} C_VEL
LIN {X 0,Y 84.393,Z 1128.895,A -85,B 0,C 180,E1 33263.693,E2 33263.693} C_VEL
LIN {X 0,Y 120.587,Z 1116.172,A -85,B 0,C 180,E1 33280.037,E2 33280.037} C_VEL
LIN {X 0,Y 157.606,Z 1099.173,A -85,B 0,C 180,E1 33288.168,E2 33288.168} C_VEL
LIN {X 0,Y 197.765,Z 1075.117,A -85,B 0,C 180,E1 33293.394,E2 33293.394} C_VEL
LIN {X 0,Y 228.919,Z 1051.358,A -85,B 0,C 180,E1 33296.21,E2 33296.21} C_VEL
LIN {X 0,Y 229.815,Z 1050.847,A -85,B 0,C 180,E1 33298.968,E2 33298.968} C_VEL
LIN {X 0,Y 193.909,Z 1078.481,A -85,B 0,C 180,E1 33302.147,E2 33302.147} C_VEL
LIN {X 0,Y 177.961,Z 1088.77,A -85,B 0,C 180,E1 33303.905,E2 33303.905} C_VEL
LIN {X 0,Y 170.513,Z 1093.144,A -85,B 0,C 180,E1 33304.438,E2 33304.438} C_VEL
LIN {X 0,Y 148.997,Z 1104.177,A -85,B 0,C 180,E1 33304.905,E2 33304.905} C_VEL
LIN {X 0,Y 147.118,Z 1105.076,A -85,B 0,C 180,E1 33305.159,E2 33305.159} C_VEL
LIN {X 0,Y 108.749,Z 1121.809,A -85,B 0,C 180,E1 33313.407,E2 33313.407} C_VEL
LIN {X 0,Y 71.248,Z 1134.042,A -85,B 0,C 180,E1 33331.952,E2 33331.952} C_VEL
LIN {X 0,Y 52.672,Z 1139.24,A -85,B 0,C 180,E1 33359.326,E2 33359.326} C_VEL
LIN {X 0,Y 48.941,Z 1141.036,A -85,B 0,C 180,E1 33389.99,E2 33389.99} C_VEL
LIN {X 0,Y 53.913,Z 1140.501,A -85,B 0,C 180,E1 33424.084,E2 33424.084} C_VEL
LIN {X 0,Y 82.871,Z 1134.928,A -85,B 0,C 180,E1 33455.729,E2 33455.729} C_VEL
LIN {X 0,Y 122.794,Z 1123.517,A -85,B 0,C 180,E1 33469.869,E2 33469.869} C_VEL
LIN {X 0,Y 162.742,Z 1107.641,A -85,B 0,C 180,E1 33476.483,E2 33476.483} C_VEL
LIN {X 0,Y 189.454,Z 1094.208,A -85,B 0,C 180,E1 33479.313,E2 33479.313} C_VEL
LIN {X 0,Y 177.565,Z 1100.238,A -85,B 0,C 180,E1 33480.848,E2 33480.848} C_VEL
LIN {X 0,Y 136.919,Z 1117.494,A -85,B 0,C 180,E1 33486.677,E2 33486.677} C_VEL
LIN {X 0,Y 95.425,Z 1129.97,A -85,B 0,C 180,E1 33498.187,E2 33498.187} C_VEL
LIN {X 0,Y 61.54,Z 1136.541,A -85,B 0,C 180,E1 33522.566,E2 33522.566} C_VEL
LIN {X 0,Y 49.577,Z 1137.779,A -85,B 0,C 180,E1 33552.264,E2 33552.264} C_VEL
LIN {X 0,Y 48.899,Z 1137.496,A -85,B 0,C 180,E1 33570.01,E2 33570.01} C_VEL
LIN {X 0,Y 56.344,Z 1135.281,A -85,B 0,C 180,E1 33602.449,E2 33602.449} C_VEL
LIN {X 0,Y 79.926,Z 1129.222,A -85,B 0,C 180,E1 33628.309,E2 33628.309} C_VEL
LIN {X 0,Y 118.093,Z 1116.532,A -85,B 0,C 180,E1 33643.692,E2 33643.692} C_VEL
LIN {X 0,Y 155.775,Z 1099.771,A -85,B 0,C 180,E1 33650.99,E2 33650.99} C_VEL
LIN {X 0,Y 197.008,Z 1075.548,A -85,B 0,C 180,E1 33655.696,E2 33655.696} C_VEL
LIN {X 0,Y 217.218,Z 1060.894,A -85,B 0,C 180,E1 33657.387,E2 33657.387} C_VEL
LIN {X 0,Y 218.354,Z 1060.06,A -85,B 0,C 180,E1 33657.841,E2 33657.841} C_VEL
LIN {X 0,Y 179.484,Z 1087.24,A -85,B 0,C 180,E1 33661.081,E2 33661.081} C_VEL
LIN {X 0,Y 147.118,Z 1105.076,A -85,B 0,C 180,E1 33665.159,E2 33665.159} C_VEL
LIN {X 0,Y 131.197,Z 1112.127,A -85,B 0,C 180,E1 33666.091,E2 33666.091} C_VEL
LIN {X 0,Y 115.012,Z 1118.411,A -85,B 0,C 180,E1 33667.28,E2 33667.28} C_VEL
LIN {X 0,Y 79.76,Z 1130.308,A -85,B 0,C 180,E1 33678.667,E2 33678.667} C_VEL
LIN {X 0,Y 51.516,Z 1137.613,A -85,B 0,C 180,E1 33702.821,E2 33702.821} C_VEL
LIN {X 0,Y 40.993,Z 1140.748,A -85,B 0,C 180,E1 33749.988,E2 33749.988} C_VEL
LIN {X 0,Y 47.442,Z 1140.228,A -85,B 0,C 180,E1 33789.557,E2 33789.557} C_VEL
LIN {X 0,Y 79.864,Z 1134.672,A -85,B 0,C 180,E1 33821.075,E2 33821.075} C_VEL
LIN {X 0,Y 121.625,Z 1123.291,A -85,B 0,C 180,E1 33833.654,E2 33833.654} C_VEL
LIN {X 0,Y 163.685,Z 1106.868,A -85,B 0,C 180,E1 33839.476,E2 33839.476} C_VEL
LIN {X 0,Y 125.16,Z 1121.461,A -85,B 0,C 180,E1 33845.136,E2 33845.136} C_VEL
LIN {X 0,Y 85.303,Z 1131.975,A -85,B 0,C 180,E1 33856.437,E2 33856.437} C_VEL
LIN {X 0,Y 56.375,Z 1136.815,A -85,B 0,C 180,E1 33876.488,E2 33876.488} C_VEL
LIN {X 0,Y 42.036,Z 1138.058,A -85,B 0,C 180,E1 33908.944,E2 33908.944} C_VEL
LIN {X 0,Y 40.96,Z 1137.783,A -85,B 0,C 180,E1 33930.012,E2 33930.012} C_VEL
LIN {X 0,Y 49.827,Z 1135.587,A -85,B 0,C 180,E1 33967.352,E2 33967.352} C_VEL
LIN {X 0,Y 76.029,Z 1129.55,A -85,B 0,C 180,E1 33993.445,E2 33993.445} C_VEL
LIN {X 0,Y 112.593,Z 1118.187,A -85,B 0,C 180,E1 34006.679,E2 34006.679} C_VEL
LIN {X 0,Y 154.143,Z 1100.466,A -85,B 0,C 180,E1 34013.842,E2 34013.842} C_VEL
LIN {X 0,Y 190.317,Z 1079.978,A -85,B 0,C 180,E1 34017.522,E2 34017.522} C_VEL
LIN {X 0,Y 151.163,Z 1102.517,A -85,B 0,C 180,E1 34021.379,E2 34021.379} C_VEL
LIN {X 0,Y 115.012,Z 1118.411,A -85,B 0,C 180,E1 34027.28,E2 34027.28} C_VEL
LIN {X 0,Y 98.604,Z 1123.923,A -85,B 0,C 180,E1 34028.885,E2 34028.885} C_VEL
LIN {X 0,Y 82.107,Z 1128.642,A -85,B 0,C 180,E1 34031.198,E2 34031.198} C_VEL
LIN {X 0,Y 46.399,Z 1137.301,A -85,B 0,C 180,E1 34055.474,E2 34055.474} C_VEL
LIN {X 0,Y 33.042,Z 1140.46,A -85,B 0,C 180,E1 34109.985,E2 34109.985} C_VEL
LIN {X 0,Y 41.541,Z 1139.955,A -85,B 0,C 180,E1 34156.661,E2 34156.661} C_VEL
LIN {X 0,Y 77.601,Z 1134.415,A -85,B 0,C 180,E1 34186.787,E2 34186.787} C_VEL
LIN {X 0,Y 120.994,Z 1123.064,A -85,B 0,C 180,E1 34197.511,E2 34197.511} C_VEL
LIN {X 0,Y 135.991,Z 1117.923,A -85,B 0,C 180,E1 34199.816,E2 34199.816} C_VEL
LIN {X 0,Y 98.846,Z 1128.834,A -85,B 0,C 180,E1 34206.485,E2 34206.485} C_VEL
LIN {X 0,Y 64.226,Z 1135.504,A -85,B 0,C 180,E1 34219.782,E2 34219.782} C_VEL
LIN {X 0,Y 36.938,Z 1138.228,A -85,B 0,C 180,E1 34254.952,E2 34254.952} C_VEL
LIN {X 0,Y 33.014,Z 1138.071,A -85,B 0,C 180,E1 34290.015,E2 34290.015} C_VEL
LIN {X 0,Y 43.771,Z 1135.894,A -85,B 0,C 180,E1 34333.682,E2 34333.682} C_VEL
LIN {X 0,Y 72.803,Z 1129.879,A -85,B 0,C 180,E1 34359.09,E2 34359.09} C_VEL
LIN {X 0,Y 114.632,Z 1117.251,A -85,B 0,C 180,E1 34371.394,E2 34371.394} C_VEL
LIN {X 0,Y 155.358,Z 1099.907,A -85,B 0,C 180,E1 34376.996,E2 34376.996} C_VEL
LIN {X 0,Y 159.336,Z 1097.882,A -85,B 0,C 180,E1 34377.392,E2 34377.392} C_VEL
LIN {X 0,Y 120.977,Z 1115.545,A -85,B 0,C 180,E1 34382.089,E2 34382.089} C_VEL
LIN {X 0,Y 82.107,Z 1128.642,A -85,B 0,C 180,E1 34391.198,E2 34391.198} C_VEL
LIN {X 0,Y 69.863,Z 1131.708,A -85,B 0,C 180,E1 34393.977,E2 34393.977} C_VEL
LIN {X 0,Y 51.008,Z 1135.312,A -85,B 0,C 180,E1 34398.779,E2 34398.779} C_VEL
LIN {X 0,Y 49.149,Z 1135.659,A -85,B 0,C 180,E1 34400.056,E2 34400.056} C_VEL
LIN {X 0,Y 27.687,Z 1139.361,A -85,B 0,C 180,E1 34436.9,E2 34436.9} C_VEL
LIN {X 0,Y 25.097,Z 1140.173,A -85,B 0,C 180,E1 34469.98,E2 34469.98} C_VEL
LIN {X 0,Y 36.472,Z 1139.682,A -85,B 0,C 180,E1 34525.936,E2 34525.936} C_VEL
LIN {X 0,Y 76.155,Z 1134.159,A -85,B 0,C 180,E1 34552.753,E2 34552.753} C_VEL
LIN {X 0,Y 107.947,Z 1126.672,A -85,B 0,C 180,E1 34560.012,E2 34560.012} C_VEL
LIN {X 0,Y 61.944,Z 1135.77,A -85,B 0,C 180,E1 34572.672,E2 34572.672} C_VEL
LIN {X 0,Y 36.565,Z 1138.295,A -85,B 0,C 180,E1 34594.281,E2 34594.281} C_VEL
LIN {X 0,Y 25.077,Z 1138.358,A -85,B 0,C 180,E1 34650.02,E2 34650.02} C_VEL
LIN {X 0,Y 38.421,Z 1136.201,A -85,B 0,C 180,E1 34701.889,E2 34701.889} C_VEL
LIN {X 0,Y 70.353,Z 1130.206,A -85,B 0,C 180,E1 34725.166,E2 34725.166} C_VEL
LIN {X 0,Y 113.709,Z 1117.611,A -85,B 0,C 180,E1 34735.39,E2 34735.39} C_VEL
LIN {X 0,Y 127.698,Z 1112.376,A -85,B 0,C 180,E1 34737.245,E2 34737.245} C_VEL
LIN {X 0,Y 90.808,Z 1125.515,A -85,B 0,C 180,E1 34743.108,E2 34743.108} C_VEL
LIN {X 0,Y 49.149,Z 1135.659,A -85,B 0,C 180,E1 34760.056,E2 34760.056} C_VEL
LIN {X 0,Y 37.46,Z 1137.485,A -85,B 0,C 180,E1 34767.513,E2 34767.513} C_VEL
LIN {X 0,Y 19.327,Z 1139.27,A -85,B 0,C 180,E1 34794.227,E2 34794.227} C_VEL
LIN {X 0,Y 17.139,Z 1139.885,A -85,B 0,C 180,E1 34829.971,E2 34829.971} C_VEL
LIN {X 0,Y 32.649,Z 1139.409,A -85,B 0,C 180,E1 34897.728,E2 34897.728} C_VEL
LIN {X 0,Y 75.56,Z 1133.902,A -85,B 0,C 180,E1 34918.91,E2 34918.91} C_VEL
LIN {X 0,Y 80.311,Z 1133.014,A -85,B 0,C 180,E1 34920.016,E2 34920.016} C_VEL
LIN {X 0,Y 46.252,Z 1137.632,A -85,B 0,C 180,E1 34931.492,E2 34931.492} C_VEL
LIN {X 0,Y 21.451,Z 1138.898,A -85,B 0,C 180,E1 34965.248,E2 34965.248} C_VEL
LIN {X 0,Y 17.125,Z 1138.646,A -85,B 0,C 180,E1 35010.029,E2 35010.029} C_VEL
LIN {X 0,Y 34.09,Z 1136.508,A -85,B 0,C 180,E1 35072.472,E2 35072.472} C_VEL
LIN {X 0,Y 68.742,Z 1130.534,A -85,B 0,C 180,E1 35091.621,E2 35091.621} C_VEL
LIN {X 0,Y 95.129,Z 1123.791,A -85,B 0,C 180,E1 35097.284,E2 35097.284} C_VEL
LIN {X 0,Y 53.736,Z 1134.134,A -85,B 0,C 180,E1 35107.405,E2 35107.405} C_VEL
LIN {X 0,Y 21.431,Z 1139.062,A -85,B 0,C 180,E1 35145.128,E2 35145.128} C_VEL
LIN {X 0,Y 19.327,Z 1139.27,A -85,B 0,C 180,E1 35154.227,E2 35154.227} C_VEL
LIN {X 0,Y 13.821,Z 1139.825,A -85,B 0,C 180,E1 35196.584,E2 35196.584} C_VEL
LIN {X 0,Y 23.331,Z 1139.41,A -85,B 0,C 180,E1 35265.805,E2 35265.805} C_VEL
LIN {X 0,Y 49.074,Z 1137.514,A -85,B 0,C 180,E1 35280.027,E2 35280.027} C_VEL
LIN {X 0,Y 16.748,Z 1139.177,A -85,B 0,C 180,E1 35305.609,E2 35305.609} C_VEL
LIN {X 0,Y 9.169,Z 1138.934,A -85,B 0,C 180,E1 35370.054,E2 35370.054} C_VEL
LIN {X 0,Y 17.725,Z 1138.149,A -85,B 0,C 180,E1 35428.543,E2 35428.543} C_VEL
LIN {X 0,Y 60.544,Z 1132.362,A -85,B 0,C 180,E1 35456.858,E2 35456.858} C_VEL
LIN {X 0,Y 30.54,Z 1137.283,A -85,B 0,C 180,E1 35468.163,E2 35468.163} C_VEL
LIN {X 0,Y 9.178,Z 1139.597,A -85,B 0,C 180,E1 35549.946,E2 35549.946} C_VEL
LIN {X 0,Y 23.331,Z 1139.41,A -85,B 0,C 180,E1 35625.805,E2 35625.805} C_VEL
LIN {X 0,Y 17.605,Z 1139.487,A -85,B 0,C 180,E1 35632.537,E2 35632.537} C_VEL
LIN {X 0,Y 11.949,Z 1138.612,A -85,B 0,C 180,E1 35453.757,E2 35453.757} C_VEL
LIN {X 0,Y 15.144,Z 1138.463,A -85,B 0,C 180,E1 35456.786,E2 35456.786} C_VEL
LIN {X 0,Y 1.213,Z 1139.309,A -85,B 0,C 180,E1 35549.59,E2 35549.59} C_VEL
LIN {X 0,Y 9.161,Z 1139.464,A -85,B 0,C 180,E1 35640.144,E2 35640.144} C_VEL
LIN {X 0,Y 11.949,Z 1138.612,A -85,B 0,C 180,E1 35813.757,E2 35813.757} C_VEL
LIN {X 0,Y 14.042,Z 1140.609,A -85,B 0,C 180,E1 35814.626,E2 35814.626} C_VEL
LIN {X 0,Y 14.042,Z 1164.5,A -85,B 0,C 180,E1 35814.626,E2 35814.626} C_VEL
LIN {X 0,Y 14.042,Z 1164.5,A -85,B 0,C 180,E1 35814.626,E2 35814.626}

